// TIA Portal project "XSFW_TIA31001_A0_V15.1" (V15.1)

(* hardware
DEVICE "S7-1200 station_1"  S7-1200 Station
   slot 0: "Rack_0"  S7-1200 Rack  Rack  V1.0
   slot 1: "PLC_Divider"  CPU 1214C DC/DC/DC  6ES7 214-1AG40-0XB0  V4.2
   slot 2: "DI 16/DQ 16x24VDC_1"  6ES7 223-1BL32-0XB0  V2.0
   slot 3: "AI 4x13BIT/AQ 2x14BIT_1"  6ES7 234-4HE32-0XB0  V2.0
   slot 101: "CM 1243-5"  CM 1243-5  6GK7 243-5DX30-0XE0  V1.3
DEVICE "CSM"  SCALANCE X-Station
   slot 0: "Bastidor SCALANCE X"  Rail
   slot 0: "Switch"  6GK7 277-1AA00-0AA0
DEVICE "HMI_1"  KTP700 Basic PN
   slot 0: "HMI_1"  KTP700 Basic PN  6AV2 123-2GB03-0AX0  15.0.0.0
   slot 1: "HMI_RT_1"  KTP700 Basic PN  6AV2 123-2GB03-0AX0  15.0.0.0
   slot 5: "HMI_1.IE_CP_1"  PROFINET Interface  15.0.0.0
      slot 1: "Interfaz PROFINET_1"  PROFINET Interface
         slot 1: "Port_1"  Port
DEVICE "Dispositivo GSD_1"  GSD.Device.PN
   slot 0: "Rack"  Rack  V1.0
   slot 0: "V90-X"  SINAMICS V90 PN V1.0  6SL3 210-5Fxxx-xxFx  V1.00
      slot 0: "SINAMICS V90 PN V1.0"  SINAMICS V90 PN V1.0
      slot 1: "PN-IO"  PN-IO
         slot 1: "Puerto 1"  Port 1
         slot 2: "Puerto 2"  Port 2
      slot 1: "Drive"  Drive
         slot 0: "Punto de acceso a módulo"  Module Access Point
         slot 1: "sin PROFIsafe"  without PROFIsafe
   slot 2: "Telegrama estándar 3, PZD-5/9"  Standard telegram 3, PZD-5/9
DEVICE "Dispositivo GSD_2"  GSD.Device.PN
   slot 0: "Rack"  Rack  V1.0
   slot 0: "V90-Y"  SINAMICS V90 PN V1.0  6SL3 210-5Fxxx-xxFx  V1.00
      slot 0: "SINAMICS V90 PN V1.0"  SINAMICS V90 PN V1.0
      slot 1: "PN-IO"  PN-IO
         slot 1: "Puerto 1"  Port 1
         slot 2: "Puerto 2"  Port 2
      slot 1: "Drive"  Drive
         slot 0: "Punto de acceso a módulo"  Module Access Point
         slot 1: "sin PROFIsafe"  without PROFIsafe
   slot 2: "Telegrama estándar 3, PZD-5/9"  Standard telegram 3, PZD-5/9
*)

// ===== PLC "PLC_Divider"  CPU 1214C DC/DC/DC =====

VAR_GLOBAL   // PLC tag table "Tabla de variables estándar"
   "iCntBot" AT %I0.3 : Bool;
   "iSnsBotBaj" AT %I0.4 : Bool;
   "iSnsBotAlt" AT %I0.5 : Bool;
   "iCH_A" AT %I0.0 : Bool;
   "iCH_B" AT %I0.1 : Bool;
   "iCH_Z" AT %I0.2 : Bool;
   "iSns_Ch1Full" AT %I2.5 : Bool;
   "iSns_Ch2Full" AT %I2.6 : Bool;
   "iSns_Ch3Full" AT %I2.7 : Bool;
   "iSign_HabInv" AT %I3.0 : Bool;
   "iPul_Marcha" AT %I3.1 : Bool;
   "iPul_Parada" AT %I3.2 : Bool;
   "iPul_Rst" AT %I3.3 : Bool;
   "iProt_Abiertas" AT %I3.4 : Bool;
   "iTrip_Inverter" AT %I3.5 : Bool;
   "iRef_Analog" AT %IW54 : Int;
   "qRev_Alarma" AT %Q0.0 : Bool;
   "qSem_Verde" AT %Q0.1 : Bool;
   "qSem_rojo" AT %Q0.2 : Bool;
   "qTest_Marcha" AT %Q0.3 : Bool;
   "qRes_Alarma" AT %Q0.4 : Bool;
   "qRes_Inversor" AT %Q0.5 : Bool;
   "qFwd_Inversor" AT %Q0.6 : Bool;
   "qTrig_2" AT %Q0.7 : Bool;
   "qSign_Marcha" AT %Q1.0 : Bool;
   "qSign_Falla" AT %Q1.1 : Bool;
   "qTrig_1" AT %Q2.0 : Bool;
   "qTrig_22" AT %Q2.1 : Bool;
   "qRef_Analog" AT %IW82 : Int;
   "System_Byte" AT %MB1 : Byte;
   "FirstScan" AT %M1.0 : Bool;
   "DiagStatusUpdate" AT %M1.1 : Bool;
   "AlwaysTRUE" AT %M1.2 : Bool;
   "AlwaysFALSE" AT %M1.3 : Bool;
   "Clock_Byte" AT %MB0 : Byte;
   "Clock_10Hz" AT %M0.0 : Bool;
   "Clock_5Hz" AT %M0.1 : Bool;
   "Clock_2.5Hz" AT %M0.2 : Bool;
   "Clock_2Hz" AT %M0.3 : Bool;
   "Clock_1.25Hz" AT %M0.4 : Bool;
   "Clock_1Hz" AT %M0.5 : Bool;
   "Clock_0.625Hz" AT %M0.6 : Bool;
   "Clock_0.5Hz" AT %M0.7 : Bool;
   "Trip_Inverter" AT %M100.2 : Bool;
   "Marca_Homing" AT %M102.1 : Bool;
   "Eje_X_Drive_IN" AT %I68.0 : "PD_TEL1_IN";
   "Eje_X_Drive_OUT" AT %Q84.0 : "PD_TEL1_OUT";
   "Eje_X_Encoder_IN" AT %I68.0 : "PD_TEL81_IN";
   "Eje_X_Encoder_OUT" AT %Q84.0 : "PD_TEL81_OUT";
   "Eje_Y_Drive_IN" AT %I104.0 : "PD_TEL3_IN";
   "Eje_Y_Drive_OUT" AT %Q74.0 : "PD_TEL3_OUT";
   "Eje_1_Drive_IN" AT %I68.0 : "PD_TEL3_IN";
   "Eje_1_Drive_OUT" AT %Q64.0 : "PD_TEL3_OUT";
END_VAR

VAR_GLOBAL   // PLC tag table "Alarmas"
   "Alarmas_1" AT %MW100 : Word;
   "ProteccionAbierta" AT %M100.0 : Bool;   // Señal I3.4 en 1
   "BotellaCaida" AT %M100.1 : Bool;
END_VAR

VAR_GLOBAL   // PLC tag table "Inicializaciòn"
   "Marcas para la inicializaciòn" AT %MW102 : Word;
   "Start" AT %M102.0 : Bool;
END_VAR

DATA_BLOCK "01_LINEA_Entradas-DB"   // DB1
{ S7_Optimized_Access := 'TRUE' }
VERSION : 0.1
   VAR
      Contador : Bool;   // Pulsador de marcha
      Sensor_Bajo : Bool;   // Pulsador de parada
      Sensor_Alto : Bool;   // Pulsador de marcha columna 4
      CH_A : Bool;   // Pulsador de parada de emergancia columna 4
      CH_B : Bool;   // Pulsador de marcha columna 6
      CH_Z : Bool;   // Pulsador de parada de emergancia columna 6
      Canal1_Full : Bool;   // Pulsador de marcha columna 9
      Canal2_Full : Bool;   // Pulsador de parada de emergancia columna 9
      Canal3_Full : Bool;   // Pulsador de marcha columna 11
      Hab_Inverter : Bool;   // Pulsador de parada de emergancia columna 11
      Marcha : Bool;   // Pulsador de marcha columna 12
      Parada : Bool;   // Pulsador de parada de emergancia columna 12
      Reset : Bool;   // Pulsador de parada de emergancia del tablero general
      Protecciones_Abiertas : Bool;   // Pulsador de parada de emergencia del tablero de la fosa
      Trip_Inverter : Bool;   // Señal de falla del variador
   END_VAR
BEGIN
END_DATA_BLOCK

DATA_BLOCK "02_LINEA_Salidas-DB"   // DB2
{ S7_Optimized_Access := 'TRUE' }
VERSION : 0.1
   VAR
      Alarma_Sonora : Bool;   // Marcha para el variador
      Semaforo_Verde : Bool;   // Sentido adelante variador
      Semaforo_Rojo : Bool;   // Sentido atras variador
      Testigo_Marcha : Bool;   // Indicador sonoro
      Reset_Alarma : Bool;   // Indicador de linea en marcha
      Reset_Inverter : Bool;   // Indicador de linea parada
      Avance_Inverter : Bool;   // Buzzer de la baliza del tablero principal
      Trigger_2 : Bool;   // Lampara verde de la baliza del tablero principal
      EnMarcha : Bool;   // Lampara roja de la baliza del tablero principal
      EnFalla : Bool;   // Lampara amarilla de la baliza del tablero principal
      Trigger_11 : Bool;
      Trigger_22 : Bool;
      Ref_20mA : Int;
   END_VAR
BEGIN
END_DATA_BLOCK

DATA_BLOCK "MotorInverter"   // DB5
{ S7_Optimized_Access := 'TRUE' }
VERSION : 0.1
// stored: InstanceOfName Motor Simple
"Motor Simple"
BEGIN
END_DATA_BLOCK

DATA_BLOCK "Cuentas_Matematicas1_DB"   // DB15
{ S7_Optimized_Access := 'TRUE' }
VERSION : 0.1
   VAR
      MovXNeg : Real := 0.0;
      Mov2X : Real := 0.0;
      Mov2XNeg : Real := 0.0;
      MovYNeg : Real := 0.0;
   END_VAR
BEGIN
END_DATA_BLOCK

DATA_BLOCK "FB_GENERAL_DB"   // DB17
{ S7_Optimized_Access := 'FALSE' }
VERSION : 0.1
// stored: InstanceOfName FB_GENERAL
"FB_GENERAL"
BEGIN
END_DATA_BLOCK

DATA_BLOCK "DB_GENERAL"   // DB100
{ S7_Optimized_Access := 'FALSE' }
VERSION : 0.1
// stored: InstanceOfName FB_GENERAL
"FB_GENERAL"
BEGIN
END_DATA_BLOCK

// folder: COMANDOS

DATA_BLOCK "DB_SUB_0_COM_GENERAL"   // DB600
{ S7_Optimized_Access := 'FALSE' }
VERSION : 0.1
   VAR
      ManipEsperaCarro : Bool;
      RecepCarroConfir : Bool;
      SalidaEsperaCarro1 : Bool;
      SalidaEsperaCarro2 : Bool;
      TengoCarroEnPortacarro : Bool;
      ReconocimientoAlarmas : Bool;
   END_VAR
BEGIN
END_DATA_BLOCK

// folder: INCIDENTES

DATA_BLOCK "DB_INC_GENERAL"   // DB500
{ S7_Optimized_Access := 'FALSE' }
VERSION : 0.1
// stored: InstanceOfName FB_INC_GENERAL
"FB_INC_GENERAL"
BEGIN
END_DATA_BLOCK

// folder: PUESTA EN MARCHA

DATA_BLOCK "DB_PUESTA_MARCHA"   // DB10
{ S7_Optimized_Access := 'TRUE' }
VERSION : 0.1
   VAR
      MovYmm : Real;
      MovXmm : Real;
      TChFull : Time := T#1S;
   END_VAR
BEGIN
END_DATA_BLOCK

// folder: System blocks/Program resources

DATA_BLOCK "IEC_Counter_0_DB"   // DB6
{ S7_Optimized_Access := 'TRUE' }
AUTHOR : Simatic
FAMILY : IEC
NAME : CNTR
VERSION : 1.0
// stored: InstanceOfName IEC_COUNTER
"IEC_COUNTER"
BEGIN
END_DATA_BLOCK

DATA_BLOCK "IEC_Timer_0_DB"   // DB7
{ S7_Optimized_Access := 'TRUE' }
AUTHOR : Simatic
FAMILY : IEC
NAME : IEC_TMR
VERSION : 1.0
// stored: InstanceOfName IEC_TIMER
"IEC_TIMER"
BEGIN
END_DATA_BLOCK

DATA_BLOCK "IEC_Counter_1_DB"   // DB8
{ S7_Optimized_Access := 'TRUE' }
AUTHOR : Simatic
FAMILY : IEC
NAME : CNTR
VERSION : 1.0
// stored: InstanceOfName IEC_COUNTER
"IEC_COUNTER"
BEGIN
END_DATA_BLOCK

DATA_BLOCK "IEC_Counter_2_DB"   // DB9
{ S7_Optimized_Access := 'TRUE' }
AUTHOR : Simatic
FAMILY : IEC
NAME : CNTR
VERSION : 1.0
// stored: InstanceOfName IEC_COUNTER
"IEC_COUNTER"
BEGIN
END_DATA_BLOCK

DATA_BLOCK "IEC_Timer_ChFull"   // DB11
{ S7_Optimized_Access := 'TRUE' }
AUTHOR : Simatic
FAMILY : IEC
NAME : IEC_TMR
VERSION : 1.0
// stored: InstanceOfName IEC_TIMER
"IEC_TIMER"
BEGIN
END_DATA_BLOCK

// folder: VISUALIZACION

DATA_BLOCK "DB_VIS_GENERAL"   // DB800
{ S7_Optimized_Access := 'FALSE' }
VERSION : 0.1
   VAR
      CantBot : Int;
      AlarmaProtecciòn : Bool;
      AlarmaBotellaCaida : Bool;
      Homing : Bool;
   END_VAR
BEGIN
END_DATA_BLOCK

// folder: (top level)

DATA_BLOCK "Eje_Y"   // DB4, Motion_DB
{ S7_Optimized_Access := 'TRUE' }
AUTHOR : SIMATIC
FAMILY : BasicMC
NAME : TO_PosAx
VERSION : 6.0
// stored: InstanceOfName TO_PositioningAxis
"TO_PositioningAxis"
BEGIN
   // Axis.Encoder.TelegramAddressOutCU = %Q74.0
   // Axis.Encoder.TelegramAddressInCU = %I104.0
   // Axis.Encoder.DoNameCU = V90-Y.Drive_Encóder1
   // Axis.Drive.TelegramAddressOutCU = %Q74.0
   // Axis.Drive.TelegramAddressInCU = %I104.0
   // Axis.Drive.TelegramType = 2
   // Axis.Drive.DoNameCU = V90-Y.Drive
   // Axis.LengthUnitNormalized.Time = 1
   // Axis.LengthUnitNormalized.Distance = -2
   // Axis.Encoder.SelectedHscIndexCU = -1
   // Axis.Encoder.DbTypeCU = Classic
   // Axis.Drive.DbTypeCU = Classic
END_DATA_BLOCK

DATA_BLOCK "Eje_X"   // DB12, Motion_DB
{ S7_Optimized_Access := 'TRUE' }
AUTHOR : SIMATIC
FAMILY : BasicMC
NAME : TO_PosAx
VERSION : 6.0
// stored: InstanceOfName TO_PositioningAxis
"TO_PositioningAxis"
BEGIN
   // Axis.Encoder.TelegramAddressOutCU = %Q64.0
   // Axis.Encoder.TelegramAddressInCU = %I68.0
   // Axis.Encoder.DoNameCU = V90-X.Drive_Encóder1
   // Axis.Drive.TelegramAddressOutCU = %Q64.0
   // Axis.Drive.TelegramAddressInCU = %I68.0
   // Axis.Drive.TelegramType = 2
   // Axis.Drive.DoNameCU = V90-X.Drive
   // Axis.LengthUnitNormalized.Distance = 1013
   // Axis.Encoder.SelectedHscIndexCU = -1
   // Axis.Encoder.DbTypeCU = Classic
   // Axis.Drive.DbTypeCU = Classic
END_DATA_BLOCK

FUNCTION_BLOCK "Cuentas_Matematicas1"   // FB1, LAD
{ S7_Optimized_Access := 'TRUE' }
VERSION : 0.1
BEGIN

REGION Network 1: Movimiento negativo en X
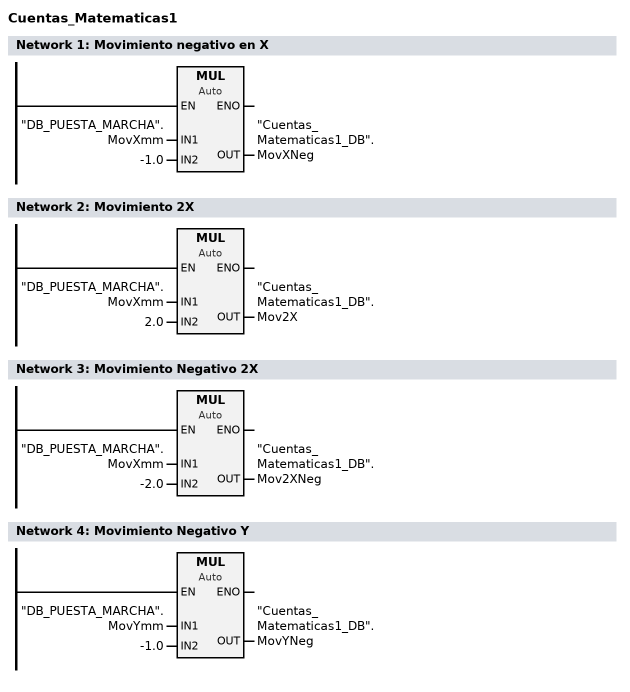
   RUNG wire#powerrail
      Mul(in1 := "DB_PUESTA_MARCHA".MovXmm, in2 := -1.0, out => "Cuentas_Matematicas1_DB".MovXNeg)
   END_RUNG
   // the same network as SCL:
   "Cuentas_Matematicas1_DB".MovXNeg := "DB_PUESTA_MARCHA".MovXmm * (-1.0);
END_REGION

REGION Network 2: Movimiento 2X
   RUNG wire#powerrail
      Mul(in1 := "DB_PUESTA_MARCHA".MovXmm, in2 := 2.0, out => "Cuentas_Matematicas1_DB".Mov2X)
   END_RUNG
   // the same network as SCL:
   "Cuentas_Matematicas1_DB".Mov2X := "DB_PUESTA_MARCHA".MovXmm * 2.0;
END_REGION

REGION Network 3: Movimiento Negativo 2X
   RUNG wire#powerrail
      Mul(in1 := "DB_PUESTA_MARCHA".MovXmm, in2 := -2.0, out => "Cuentas_Matematicas1_DB".Mov2XNeg)
   END_RUNG
   // the same network as SCL:
   "Cuentas_Matematicas1_DB".Mov2XNeg := "DB_PUESTA_MARCHA".MovXmm * (-2.0);
END_REGION

REGION Network 4: Movimiento Negativo Y
   RUNG wire#powerrail
      Mul(in1 := "DB_PUESTA_MARCHA".MovYmm, in2 := -1.0, out => "Cuentas_Matematicas1_DB".MovYNeg)
   END_RUNG
   // the same network as SCL:
   "Cuentas_Matematicas1_DB".MovYNeg := "DB_PUESTA_MARCHA".MovYmm * (-1.0);
END_REGION
END_FUNCTION_BLOCK

FUNCTION_BLOCK "FB_GENERAL"   // FB100, LAD
{ S7_Optimized_Access := 'FALSE' }
VERSION : 0.1
   VAR_OUTPUT
      DoneX : Bool;
      DoneY : Bool;
      Done2X : Bool;
      DoneHomeX : Bool;
      DoneHomeY : Bool;
   END_VAR
   VAR
      Estados : Array[0..32] of Bool;
      Concatenadoras : Array[0..32] of Bool;
      Prioritarias : Array[0..32] of Bool;
      Error_Concatenadoras : Bool;
      Error_Prioritarias : Bool;
      Cuenta_1 : Bool;
      Cuenta_2 : Bool;
      Cuenta_3 : Bool;
      "Cont_Botellas/2" : Int;
   END_VAR
BEGIN

REGION Network 1: Inicializaciòn
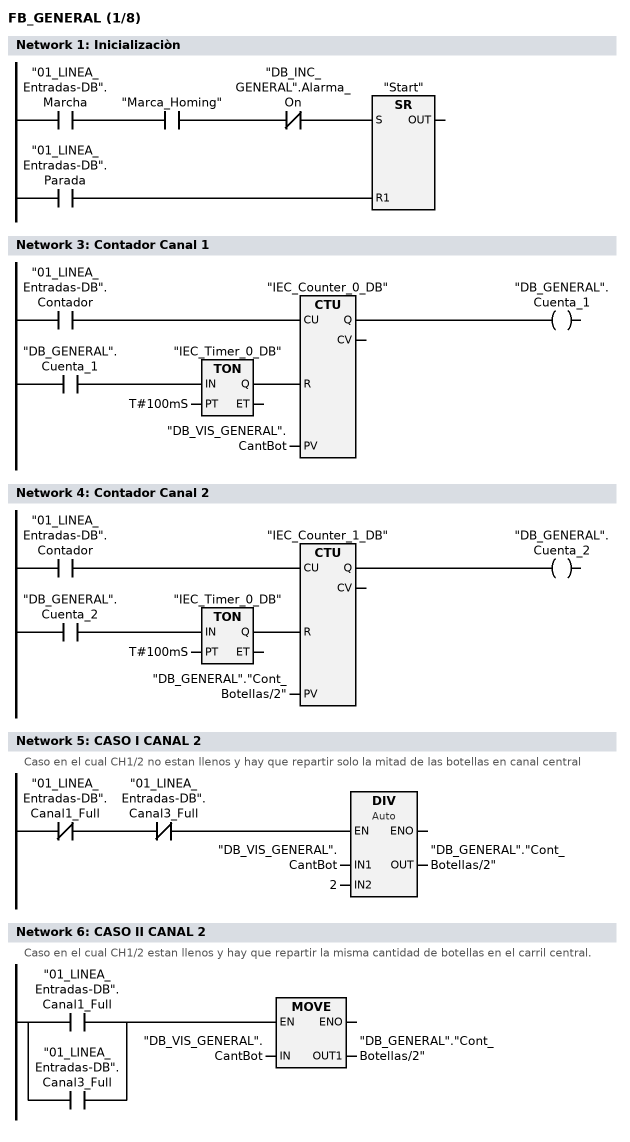
   RUNG wire#powerrail
      Contact( "01_LINEA_Entradas-DB".Marcha )
      Contact( "Marca_Homing" )
      I_Contact( "DB_INC_GENERAL".Alarma_On )
      S_SR(operand := "Start", r1 := wire#w1)
   END_RUNG
   RUNG wire#powerrail
      Contact( "01_LINEA_Entradas-DB".Parada )
   END_RUNG wire#w1
   // the same network as SCL:
   IF "01_LINEA_Entradas-DB".Marcha AND "Marca_Homing" AND NOT "DB_INC_GENERAL".Alarma_On THEN
       "Start" := TRUE;   // SR flip-flop
   END_IF;
   IF "01_LINEA_Entradas-DB".Parada THEN "Start" := FALSE; END_IF;
END_REGION

REGION Network 2: -----------------OTROS---------------
END_REGION

REGION Network 3: Contador Canal 1
   "IEC_Timer_0_DB".TON(IN := "DB_GENERAL".Cuenta_1, PT := T#100mS);
   "IEC_Counter_0_DB".CTU(CU := "01_LINEA_Entradas-DB".Contador,
                          R := "IEC_Timer_0_DB".Q,
                          PV := "DB_VIS_GENERAL".CantBot);
   "DB_GENERAL".Cuenta_1 := "IEC_Counter_0_DB".Q;
END_REGION

REGION Network 4: Contador Canal 2
   "IEC_Timer_0_DB".TON(IN := "DB_GENERAL".Cuenta_2, PT := T#100mS);
   "IEC_Counter_1_DB".CTU(CU := "01_LINEA_Entradas-DB".Contador,
                          R := "IEC_Timer_0_DB".Q,
                          PV := "DB_GENERAL"."Cont_Botellas/2");
   "DB_GENERAL".Cuenta_2 := "IEC_Counter_1_DB".Q;
END_REGION

REGION Network 5: CASO I CANAL 2
   // Caso en el cual CH1/2 no estan llenos y hay que repartir solo la mitad de las botellas en canal central
   RUNG wire#powerrail
      I_Contact( "01_LINEA_Entradas-DB".Canal1_Full )
      I_Contact( "01_LINEA_Entradas-DB".Canal3_Full )
      Div(in1 := "DB_VIS_GENERAL".CantBot, in2 := 2, out => "DB_GENERAL"."Cont_Botellas/2")
   END_RUNG
   // the same network as SCL:
   IF NOT "01_LINEA_Entradas-DB".Canal1_Full AND NOT "01_LINEA_Entradas-DB".Canal3_Full THEN
       "DB_GENERAL"."Cont_Botellas/2" := "DB_VIS_GENERAL".CantBot / 2;
   END_IF;
END_REGION

REGION Network 6: CASO II CANAL 2
   // Caso en el cual CH1/2 estan llenos y hay que repartir la misma cantidad de botellas en el carril central.
   RUNG wire#powerrail
      Contact( "01_LINEA_Entradas-DB".Canal1_Full )
      wire#w1
      Move(in := "DB_VIS_GENERAL".CantBot, out1 => "DB_GENERAL"."Cont_Botellas/2")
   END_RUNG
   RUNG wire#powerrail
      Contact( "01_LINEA_Entradas-DB".Canal3_Full )
   END_RUNG wire#w1
   // the same network as SCL:
   IF "01_LINEA_Entradas-DB".Canal1_Full OR "01_LINEA_Entradas-DB".Canal3_Full THEN
       "DB_GENERAL"."Cont_Botellas/2" := "DB_VIS_GENERAL".CantBot;
   END_IF;
END_REGION

REGION Network 7: Contador Canal 3
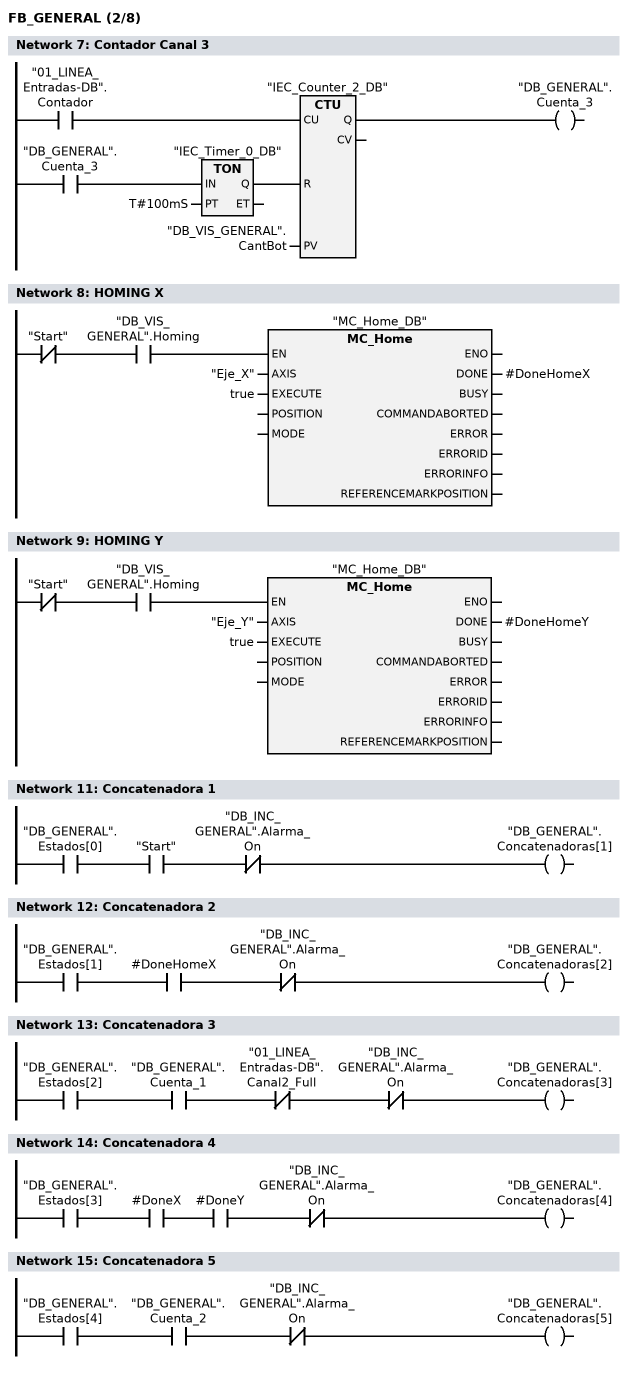
   "IEC_Timer_0_DB".TON(IN := "DB_GENERAL".Cuenta_3, PT := T#100mS);
   "IEC_Counter_2_DB".CTU(CU := "01_LINEA_Entradas-DB".Contador,
                          R := "IEC_Timer_0_DB".Q,
                          PV := "DB_VIS_GENERAL".CantBot);
   "DB_GENERAL".Cuenta_3 := "IEC_Counter_2_DB".Q;
END_REGION

REGION Network 8: HOMING X
   IF NOT "Start" AND "DB_VIS_GENERAL".Homing THEN
       "MC_Home_DB"(Axis := "Eje_X", Execute := true, Done => #DoneHomeX);   // MC_Home
   END_IF;
END_REGION

REGION Network 9: HOMING Y
   IF NOT "Start" AND "DB_VIS_GENERAL".Homing THEN
       "MC_Home_DB"(Axis := "Eje_Y", Execute := true, Done => #DoneHomeY);   // MC_Home
   END_IF;
END_REGION

REGION Network 10: --------------------Maquina de estados - 3 carriles-----------------
END_REGION

REGION Network 11: Concatenadora 1
   RUNG wire#powerrail
      Contact( "DB_GENERAL".Estados[0] )
      Contact( "Start" )
      I_Contact( "DB_INC_GENERAL".Alarma_On )
      Coil( "DB_GENERAL".Concatenadoras[1] )
   END_RUNG
   // the same network as SCL:
   "DB_GENERAL".Concatenadoras[1] := "DB_GENERAL".Estados[0] AND "Start" AND NOT "DB_INC_GENERAL".Alarma_On;
END_REGION

REGION Network 12: Concatenadora 2
   RUNG wire#powerrail
      Contact( "DB_GENERAL".Estados[1] )
      Contact( #DoneHomeX )
      I_Contact( "DB_INC_GENERAL".Alarma_On )
      Coil( "DB_GENERAL".Concatenadoras[2] )
   END_RUNG
   // the same network as SCL:
   "DB_GENERAL".Concatenadoras[2] := "DB_GENERAL".Estados[1] AND #DoneHomeX AND NOT "DB_INC_GENERAL".Alarma_On;
END_REGION

REGION Network 13: Concatenadora 3
   RUNG wire#powerrail
      Contact( "DB_GENERAL".Estados[2] )
      Contact( "DB_GENERAL".Cuenta_1 )
      I_Contact( "01_LINEA_Entradas-DB".Canal2_Full )
      I_Contact( "DB_INC_GENERAL".Alarma_On )
      Coil( "DB_GENERAL".Concatenadoras[3] )
   END_RUNG
   // the same network as SCL:
   "DB_GENERAL".Concatenadoras[3] := "DB_GENERAL".Estados[2] AND "DB_GENERAL".Cuenta_1 AND NOT "01_LINEA_Entradas-DB".Canal2_Full AND NOT "DB_INC_GENERAL".Alarma_On;
END_REGION

REGION Network 14: Concatenadora 4
   RUNG wire#powerrail
      Contact( "DB_GENERAL".Estados[3] )
      Contact( #DoneX )
      Contact( #DoneY )
      I_Contact( "DB_INC_GENERAL".Alarma_On )
      Coil( "DB_GENERAL".Concatenadoras[4] )
   END_RUNG
   // the same network as SCL:
   "DB_GENERAL".Concatenadoras[4] := "DB_GENERAL".Estados[3] AND #DoneX AND #DoneY AND NOT "DB_INC_GENERAL".Alarma_On;
END_REGION

REGION Network 15: Concatenadora 5
   RUNG wire#powerrail
      Contact( "DB_GENERAL".Estados[4] )
      Contact( "DB_GENERAL".Cuenta_2 )
      I_Contact( "DB_INC_GENERAL".Alarma_On )
      Coil( "DB_GENERAL".Concatenadoras[5] )
   END_RUNG
   // the same network as SCL:
   "DB_GENERAL".Concatenadoras[5] := "DB_GENERAL".Estados[4] AND "DB_GENERAL".Cuenta_2 AND NOT "DB_INC_GENERAL".Alarma_On;
END_REGION

REGION Network 16: Concatenadora 6
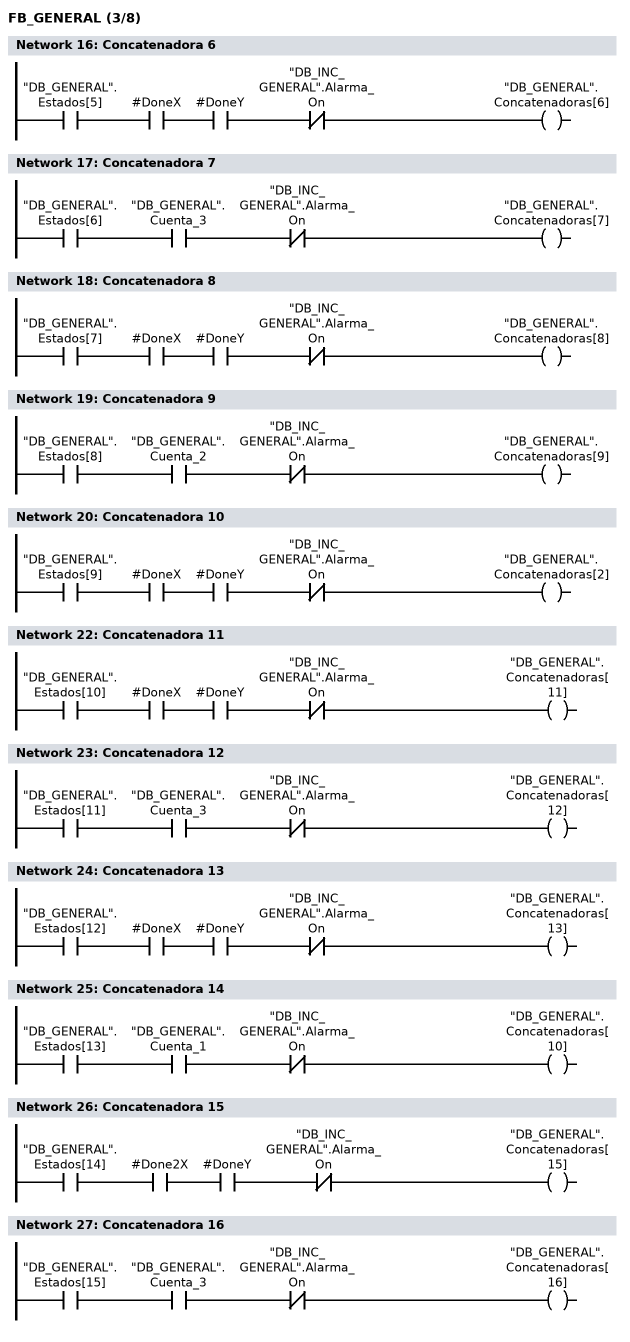
   RUNG wire#powerrail
      Contact( "DB_GENERAL".Estados[5] )
      Contact( #DoneX )
      Contact( #DoneY )
      I_Contact( "DB_INC_GENERAL".Alarma_On )
      Coil( "DB_GENERAL".Concatenadoras[6] )
   END_RUNG
   // the same network as SCL:
   "DB_GENERAL".Concatenadoras[6] := "DB_GENERAL".Estados[5] AND #DoneX AND #DoneY AND NOT "DB_INC_GENERAL".Alarma_On;
END_REGION

REGION Network 17: Concatenadora 7
   RUNG wire#powerrail
      Contact( "DB_GENERAL".Estados[6] )
      Contact( "DB_GENERAL".Cuenta_3 )
      I_Contact( "DB_INC_GENERAL".Alarma_On )
      Coil( "DB_GENERAL".Concatenadoras[7] )
   END_RUNG
   // the same network as SCL:
   "DB_GENERAL".Concatenadoras[7] := "DB_GENERAL".Estados[6] AND "DB_GENERAL".Cuenta_3 AND NOT "DB_INC_GENERAL".Alarma_On;
END_REGION

REGION Network 18: Concatenadora 8
   RUNG wire#powerrail
      Contact( "DB_GENERAL".Estados[7] )
      Contact( #DoneX )
      Contact( #DoneY )
      I_Contact( "DB_INC_GENERAL".Alarma_On )
      Coil( "DB_GENERAL".Concatenadoras[8] )
   END_RUNG
   // the same network as SCL:
   "DB_GENERAL".Concatenadoras[8] := "DB_GENERAL".Estados[7] AND #DoneX AND #DoneY AND NOT "DB_INC_GENERAL".Alarma_On;
END_REGION

REGION Network 19: Concatenadora 9
   RUNG wire#powerrail
      Contact( "DB_GENERAL".Estados[8] )
      Contact( "DB_GENERAL".Cuenta_2 )
      I_Contact( "DB_INC_GENERAL".Alarma_On )
      Coil( "DB_GENERAL".Concatenadoras[9] )
   END_RUNG
   // the same network as SCL:
   "DB_GENERAL".Concatenadoras[9] := "DB_GENERAL".Estados[8] AND "DB_GENERAL".Cuenta_2 AND NOT "DB_INC_GENERAL".Alarma_On;
END_REGION

REGION Network 20: Concatenadora 10
   RUNG wire#powerrail
      Contact( "DB_GENERAL".Estados[9] )
      Contact( #DoneX )
      Contact( #DoneY )
      I_Contact( "DB_INC_GENERAL".Alarma_On )
      Coil( "DB_GENERAL".Concatenadoras[2] )
   END_RUNG
   // the same network as SCL:
   "DB_GENERAL".Concatenadoras[2] := "DB_GENERAL".Estados[9] AND #DoneX AND #DoneY AND NOT "DB_INC_GENERAL".Alarma_On;
END_REGION

REGION Network 21: ---------------Maquina de estado - 2 carriles -------------
END_REGION

REGION Network 22: Concatenadora 11
   RUNG wire#powerrail
      Contact( "DB_GENERAL".Estados[10] )
      Contact( #DoneX )
      Contact( #DoneY )
      I_Contact( "DB_INC_GENERAL".Alarma_On )
      Coil( "DB_GENERAL".Concatenadoras[11] )
   END_RUNG
   // the same network as SCL:
   "DB_GENERAL".Concatenadoras[11] := "DB_GENERAL".Estados[10] AND #DoneX AND #DoneY AND NOT "DB_INC_GENERAL".Alarma_On;
END_REGION

REGION Network 23: Concatenadora 12
   RUNG wire#powerrail
      Contact( "DB_GENERAL".Estados[11] )
      Contact( "DB_GENERAL".Cuenta_3 )
      I_Contact( "DB_INC_GENERAL".Alarma_On )
      Coil( "DB_GENERAL".Concatenadoras[12] )
   END_RUNG
   // the same network as SCL:
   "DB_GENERAL".Concatenadoras[12] := "DB_GENERAL".Estados[11] AND "DB_GENERAL".Cuenta_3 AND NOT "DB_INC_GENERAL".Alarma_On;
END_REGION

REGION Network 24: Concatenadora 13
   RUNG wire#powerrail
      Contact( "DB_GENERAL".Estados[12] )
      Contact( #DoneX )
      Contact( #DoneY )
      I_Contact( "DB_INC_GENERAL".Alarma_On )
      Coil( "DB_GENERAL".Concatenadoras[13] )
   END_RUNG
   // the same network as SCL:
   "DB_GENERAL".Concatenadoras[13] := "DB_GENERAL".Estados[12] AND #DoneX AND #DoneY AND NOT "DB_INC_GENERAL".Alarma_On;
END_REGION

REGION Network 25: Concatenadora 14
   RUNG wire#powerrail
      Contact( "DB_GENERAL".Estados[13] )
      Contact( "DB_GENERAL".Cuenta_1 )
      I_Contact( "DB_INC_GENERAL".Alarma_On )
      Coil( "DB_GENERAL".Concatenadoras[10] )
   END_RUNG
   // the same network as SCL:
   "DB_GENERAL".Concatenadoras[10] := "DB_GENERAL".Estados[13] AND "DB_GENERAL".Cuenta_1 AND NOT "DB_INC_GENERAL".Alarma_On;
END_REGION

REGION Network 26: Concatenadora 15
   RUNG wire#powerrail
      Contact( "DB_GENERAL".Estados[14] )
      Contact( #Done2X )
      Contact( #DoneY )
      I_Contact( "DB_INC_GENERAL".Alarma_On )
      Coil( "DB_GENERAL".Concatenadoras[15] )
   END_RUNG
   // the same network as SCL:
   "DB_GENERAL".Concatenadoras[15] := "DB_GENERAL".Estados[14] AND #Done2X AND #DoneY AND NOT "DB_INC_GENERAL".Alarma_On;
END_REGION

REGION Network 27: Concatenadora 16
   RUNG wire#powerrail
      Contact( "DB_GENERAL".Estados[15] )
      Contact( "DB_GENERAL".Cuenta_3 )
      I_Contact( "DB_INC_GENERAL".Alarma_On )
      Coil( "DB_GENERAL".Concatenadoras[16] )
   END_RUNG
   // the same network as SCL:
   "DB_GENERAL".Concatenadoras[16] := "DB_GENERAL".Estados[15] AND "DB_GENERAL".Cuenta_3 AND NOT "DB_INC_GENERAL".Alarma_On;
END_REGION

REGION Network 28: Concatenadora 17
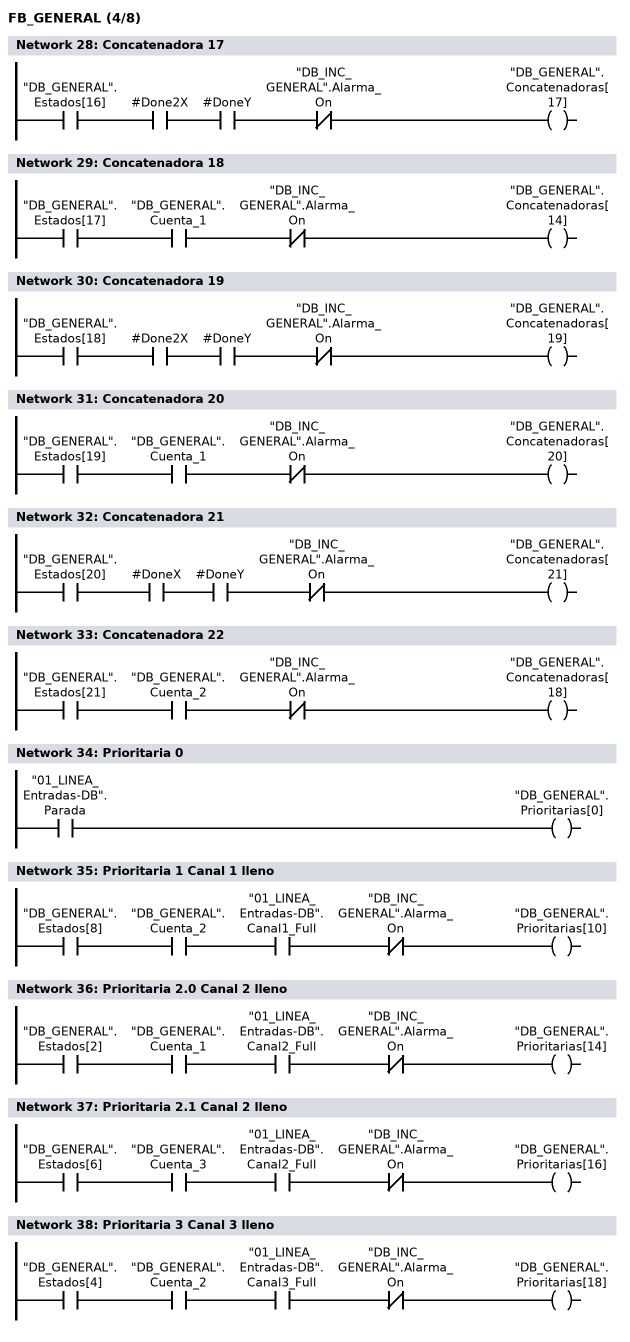
   RUNG wire#powerrail
      Contact( "DB_GENERAL".Estados[16] )
      Contact( #Done2X )
      Contact( #DoneY )
      I_Contact( "DB_INC_GENERAL".Alarma_On )
      Coil( "DB_GENERAL".Concatenadoras[17] )
   END_RUNG
   // the same network as SCL:
   "DB_GENERAL".Concatenadoras[17] := "DB_GENERAL".Estados[16] AND #Done2X AND #DoneY AND NOT "DB_INC_GENERAL".Alarma_On;
END_REGION

REGION Network 29: Concatenadora 18
   RUNG wire#powerrail
      Contact( "DB_GENERAL".Estados[17] )
      Contact( "DB_GENERAL".Cuenta_1 )
      I_Contact( "DB_INC_GENERAL".Alarma_On )
      Coil( "DB_GENERAL".Concatenadoras[14] )
   END_RUNG
   // the same network as SCL:
   "DB_GENERAL".Concatenadoras[14] := "DB_GENERAL".Estados[17] AND "DB_GENERAL".Cuenta_1 AND NOT "DB_INC_GENERAL".Alarma_On;
END_REGION

REGION Network 30: Concatenadora 19
   RUNG wire#powerrail
      Contact( "DB_GENERAL".Estados[18] )
      Contact( #Done2X )
      Contact( #DoneY )
      I_Contact( "DB_INC_GENERAL".Alarma_On )
      Coil( "DB_GENERAL".Concatenadoras[19] )
   END_RUNG
   // the same network as SCL:
   "DB_GENERAL".Concatenadoras[19] := "DB_GENERAL".Estados[18] AND #Done2X AND #DoneY AND NOT "DB_INC_GENERAL".Alarma_On;
END_REGION

REGION Network 31: Concatenadora 20
   RUNG wire#powerrail
      Contact( "DB_GENERAL".Estados[19] )
      Contact( "DB_GENERAL".Cuenta_1 )
      I_Contact( "DB_INC_GENERAL".Alarma_On )
      Coil( "DB_GENERAL".Concatenadoras[20] )
   END_RUNG
   // the same network as SCL:
   "DB_GENERAL".Concatenadoras[20] := "DB_GENERAL".Estados[19] AND "DB_GENERAL".Cuenta_1 AND NOT "DB_INC_GENERAL".Alarma_On;
END_REGION

REGION Network 32: Concatenadora 21
   RUNG wire#powerrail
      Contact( "DB_GENERAL".Estados[20] )
      Contact( #DoneX )
      Contact( #DoneY )
      I_Contact( "DB_INC_GENERAL".Alarma_On )
      Coil( "DB_GENERAL".Concatenadoras[21] )
   END_RUNG
   // the same network as SCL:
   "DB_GENERAL".Concatenadoras[21] := "DB_GENERAL".Estados[20] AND #DoneX AND #DoneY AND NOT "DB_INC_GENERAL".Alarma_On;
END_REGION

REGION Network 33: Concatenadora 22
   RUNG wire#powerrail
      Contact( "DB_GENERAL".Estados[21] )
      Contact( "DB_GENERAL".Cuenta_2 )
      I_Contact( "DB_INC_GENERAL".Alarma_On )
      Coil( "DB_GENERAL".Concatenadoras[18] )
   END_RUNG
   // the same network as SCL:
   "DB_GENERAL".Concatenadoras[18] := "DB_GENERAL".Estados[21] AND "DB_GENERAL".Cuenta_2 AND NOT "DB_INC_GENERAL".Alarma_On;
END_REGION

REGION Network 34: Prioritaria 0
   RUNG wire#powerrail
      Contact( "01_LINEA_Entradas-DB".Parada )
      Coil( "DB_GENERAL".Prioritarias[0] )
   END_RUNG
   // the same network as SCL:
   "DB_GENERAL".Prioritarias[0] := "01_LINEA_Entradas-DB".Parada;
END_REGION

REGION Network 35: Prioritaria 1 Canal 1 lleno
   RUNG wire#powerrail
      Contact( "DB_GENERAL".Estados[8] )
      Contact( "DB_GENERAL".Cuenta_2 )
      Contact( "01_LINEA_Entradas-DB".Canal1_Full )
      I_Contact( "DB_INC_GENERAL".Alarma_On )
      Coil( "DB_GENERAL".Prioritarias[10] )
   END_RUNG
   // the same network as SCL:
   "DB_GENERAL".Prioritarias[10] := "DB_GENERAL".Estados[8] AND "DB_GENERAL".Cuenta_2 AND "01_LINEA_Entradas-DB".Canal1_Full AND NOT "DB_INC_GENERAL".Alarma_On;
END_REGION

REGION Network 36: Prioritaria 2.0 Canal 2 lleno
   RUNG wire#powerrail
      Contact( "DB_GENERAL".Estados[2] )
      Contact( "DB_GENERAL".Cuenta_1 )
      Contact( "01_LINEA_Entradas-DB".Canal2_Full )
      I_Contact( "DB_INC_GENERAL".Alarma_On )
      Coil( "DB_GENERAL".Prioritarias[14] )
   END_RUNG
   // the same network as SCL:
   "DB_GENERAL".Prioritarias[14] := "DB_GENERAL".Estados[2] AND "DB_GENERAL".Cuenta_1 AND "01_LINEA_Entradas-DB".Canal2_Full AND NOT "DB_INC_GENERAL".Alarma_On;
END_REGION

REGION Network 37: Prioritaria 2.1 Canal 2 lleno
   RUNG wire#powerrail
      Contact( "DB_GENERAL".Estados[6] )
      Contact( "DB_GENERAL".Cuenta_3 )
      Contact( "01_LINEA_Entradas-DB".Canal2_Full )
      I_Contact( "DB_INC_GENERAL".Alarma_On )
      Coil( "DB_GENERAL".Prioritarias[16] )
   END_RUNG
   // the same network as SCL:
   "DB_GENERAL".Prioritarias[16] := "DB_GENERAL".Estados[6] AND "DB_GENERAL".Cuenta_3 AND "01_LINEA_Entradas-DB".Canal2_Full AND NOT "DB_INC_GENERAL".Alarma_On;
END_REGION

REGION Network 38: Prioritaria 3 Canal 3 lleno
   RUNG wire#powerrail
      Contact( "DB_GENERAL".Estados[4] )
      Contact( "DB_GENERAL".Cuenta_2 )
      Contact( "01_LINEA_Entradas-DB".Canal3_Full )
      I_Contact( "DB_INC_GENERAL".Alarma_On )
      Coil( "DB_GENERAL".Prioritarias[18] )
   END_RUNG
   // the same network as SCL:
   "DB_GENERAL".Prioritarias[18] := "DB_GENERAL".Estados[4] AND "DB_GENERAL".Cuenta_2 AND "01_LINEA_Entradas-DB".Canal3_Full AND NOT "DB_INC_GENERAL".Alarma_On;
END_REGION

REGION Network 39: Prioritaria 4 Canal 1 se vaciò
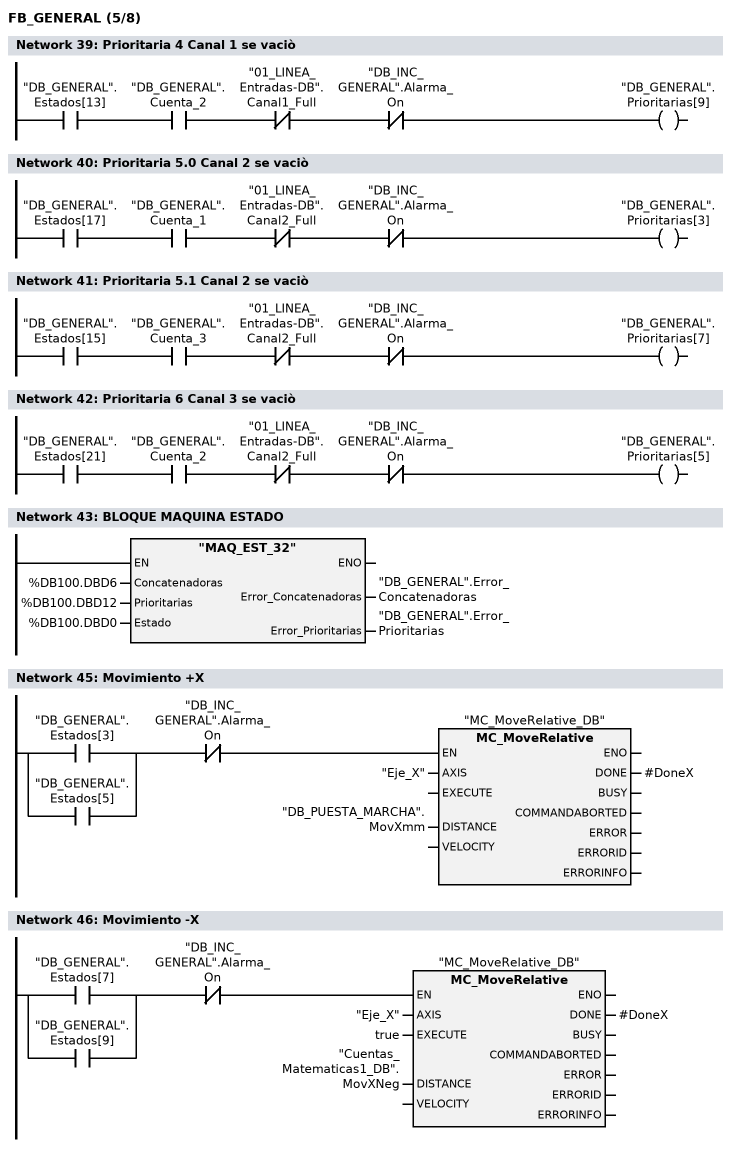
   RUNG wire#powerrail
      Contact( "DB_GENERAL".Estados[13] )
      Contact( "DB_GENERAL".Cuenta_2 )
      I_Contact( "01_LINEA_Entradas-DB".Canal1_Full )
      I_Contact( "DB_INC_GENERAL".Alarma_On )
      Coil( "DB_GENERAL".Prioritarias[9] )
   END_RUNG
   // the same network as SCL:
   "DB_GENERAL".Prioritarias[9] := "DB_GENERAL".Estados[13] AND "DB_GENERAL".Cuenta_2 AND NOT "01_LINEA_Entradas-DB".Canal1_Full AND NOT "DB_INC_GENERAL".Alarma_On;
END_REGION

REGION Network 40: Prioritaria 5.0 Canal 2 se vaciò
   RUNG wire#powerrail
      Contact( "DB_GENERAL".Estados[17] )
      Contact( "DB_GENERAL".Cuenta_1 )
      I_Contact( "01_LINEA_Entradas-DB".Canal2_Full )
      I_Contact( "DB_INC_GENERAL".Alarma_On )
      Coil( "DB_GENERAL".Prioritarias[3] )
   END_RUNG
   // the same network as SCL:
   "DB_GENERAL".Prioritarias[3] := "DB_GENERAL".Estados[17] AND "DB_GENERAL".Cuenta_1 AND NOT "01_LINEA_Entradas-DB".Canal2_Full AND NOT "DB_INC_GENERAL".Alarma_On;
END_REGION

REGION Network 41: Prioritaria 5.1 Canal 2 se vaciò
   RUNG wire#powerrail
      Contact( "DB_GENERAL".Estados[15] )
      Contact( "DB_GENERAL".Cuenta_3 )
      I_Contact( "01_LINEA_Entradas-DB".Canal2_Full )
      I_Contact( "DB_INC_GENERAL".Alarma_On )
      Coil( "DB_GENERAL".Prioritarias[7] )
   END_RUNG
   // the same network as SCL:
   "DB_GENERAL".Prioritarias[7] := "DB_GENERAL".Estados[15] AND "DB_GENERAL".Cuenta_3 AND NOT "01_LINEA_Entradas-DB".Canal2_Full AND NOT "DB_INC_GENERAL".Alarma_On;
END_REGION

REGION Network 42: Prioritaria 6 Canal 3 se vaciò
   RUNG wire#powerrail
      Contact( "DB_GENERAL".Estados[21] )
      Contact( "DB_GENERAL".Cuenta_2 )
      I_Contact( "01_LINEA_Entradas-DB".Canal2_Full )
      I_Contact( "DB_INC_GENERAL".Alarma_On )
      Coil( "DB_GENERAL".Prioritarias[5] )
   END_RUNG
   // the same network as SCL:
   "DB_GENERAL".Prioritarias[5] := "DB_GENERAL".Estados[21] AND "DB_GENERAL".Cuenta_2 AND NOT "01_LINEA_Entradas-DB".Canal2_Full AND NOT "DB_INC_GENERAL".Alarma_On;
END_REGION

REGION Network 43: BLOQUE MAQUINA ESTADO
   RUNG wire#powerrail
      "MAQ_EST_32"(Concatenadoras := %DB100.DBD6, Prioritarias := %DB100.DBD12, Estado := %DB100.DBD0, Error_Concatenadoras => "DB_GENERAL".Error_Concatenadoras, Error_Prioritarias => "DB_GENERAL".Error_Prioritarias)
   END_RUNG
   // the same network as SCL:
   "MAQ_EST_32"(Concatenadoras := %DB100.DBD6,
                Prioritarias := %DB100.DBD12,
                Estado := %DB100.DBD0,
                Error_Concatenadoras => "DB_GENERAL".Error_Concatenadoras,
                Error_Prioritarias => "DB_GENERAL".Error_Prioritarias);
END_REGION

REGION Network 44: --------------ACCIONAMIENTOS----------------
END_REGION

REGION Network 45: Movimiento +X
   IF ("DB_GENERAL".Estados[3] OR "DB_GENERAL".Estados[5]) AND NOT "DB_INC_GENERAL".Alarma_On THEN
       "MC_MoveRelative_DB"(Axis := "Eje_X", Distance := "DB_PUESTA_MARCHA".MovXmm, Done => #DoneX);   // MC_MoveRelative
   END_IF;
END_REGION

REGION Network 46: Movimiento -X
   IF ("DB_GENERAL".Estados[7] OR "DB_GENERAL".Estados[9]) AND NOT "DB_INC_GENERAL".Alarma_On THEN
       "MC_MoveRelative_DB"(Axis := "Eje_X",   // MC_MoveRelative
                            Execute := true,
                            Distance := "Cuentas_Matematicas1_DB".MovXNeg,
                            Done => #DoneX);
   END_IF;
END_REGION

REGION Network 47: Movimiento +Y
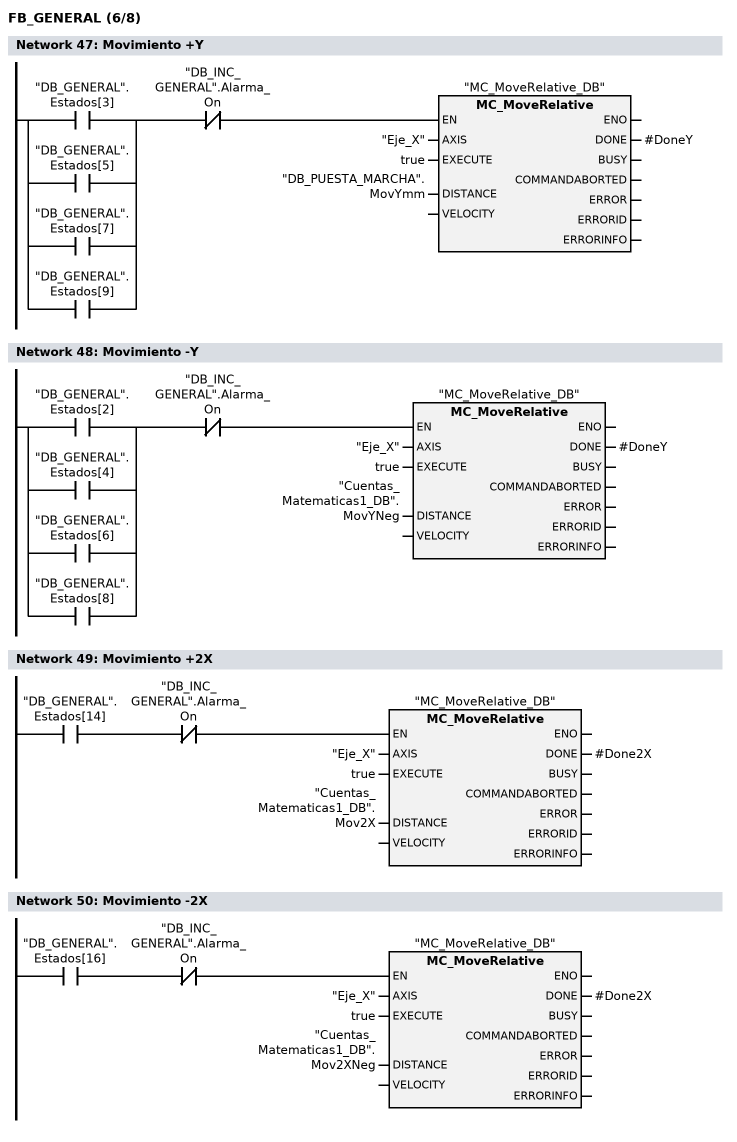
   IF ("DB_GENERAL".Estados[3] OR "DB_GENERAL".Estados[5] OR "DB_GENERAL".Estados[7] OR "DB_GENERAL".Estados[9]) AND NOT "DB_INC_GENERAL".Alarma_On THEN
       "MC_MoveRelative_DB"(Axis := "Eje_X", Execute := true, Distance := "DB_PUESTA_MARCHA".MovYmm, Done => #DoneY);   // MC_MoveRelative
   END_IF;
END_REGION

REGION Network 48: Movimiento -Y
   IF ("DB_GENERAL".Estados[2] OR "DB_GENERAL".Estados[4] OR "DB_GENERAL".Estados[6] OR "DB_GENERAL".Estados[8]) AND NOT "DB_INC_GENERAL".Alarma_On THEN
       "MC_MoveRelative_DB"(Axis := "Eje_X",   // MC_MoveRelative
                            Execute := true,
                            Distance := "Cuentas_Matematicas1_DB".MovYNeg,
                            Done => #DoneY);
   END_IF;
END_REGION

REGION Network 49: Movimiento +2X
   IF "DB_GENERAL".Estados[14] AND NOT "DB_INC_GENERAL".Alarma_On THEN
       "MC_MoveRelative_DB"(Axis := "Eje_X",   // MC_MoveRelative
                            Execute := true,
                            Distance := "Cuentas_Matematicas1_DB".Mov2X,
                            Done => #Done2X);
   END_IF;
END_REGION

REGION Network 50: Movimiento -2X
   IF "DB_GENERAL".Estados[16] AND NOT "DB_INC_GENERAL".Alarma_On THEN
       "MC_MoveRelative_DB"(Axis := "Eje_X",   // MC_MoveRelative
                            Execute := true,
                            Distance := "Cuentas_Matematicas1_DB".Mov2XNeg,
                            Done => #Done2X);
   END_IF;
END_REGION

REGION Network 51: Avance inverter
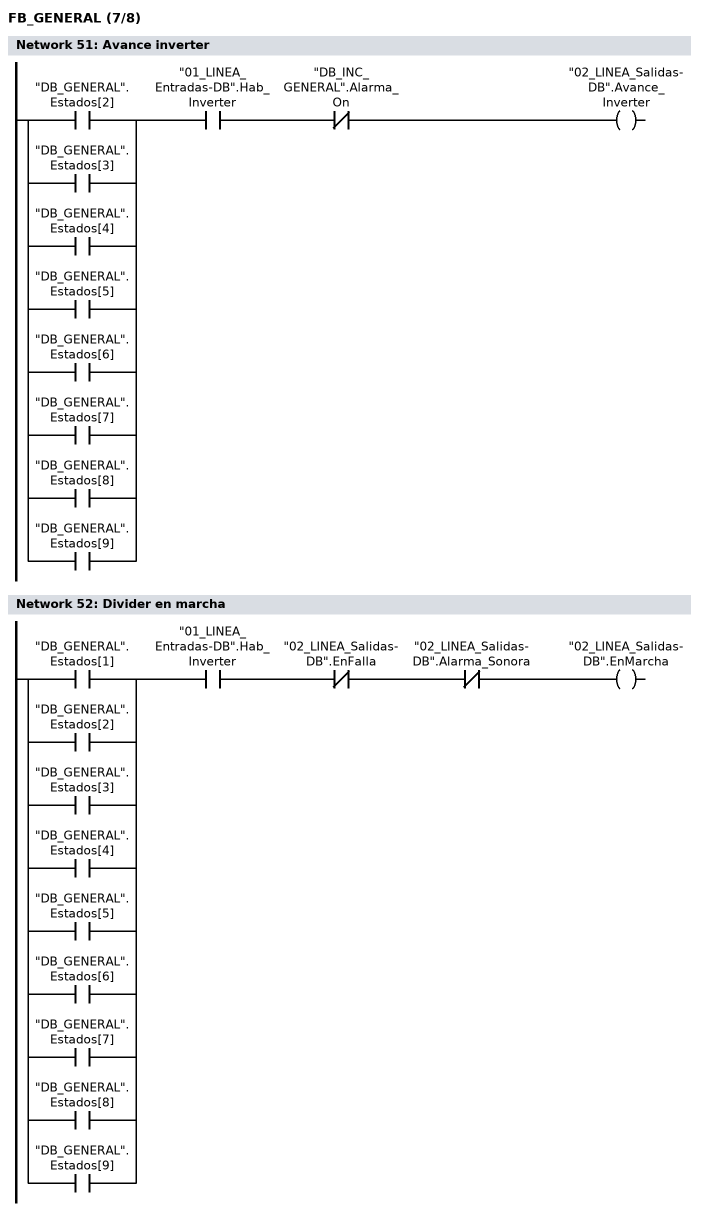
   RUNG wire#powerrail
      Contact( "DB_GENERAL".Estados[2] )
      wire#w1
      Contact( "01_LINEA_Entradas-DB".Hab_Inverter )
      I_Contact( "DB_INC_GENERAL".Alarma_On )
      Coil( "02_LINEA_Salidas-DB".Avance_Inverter )
   END_RUNG
   RUNG wire#powerrail
      Contact( "DB_GENERAL".Estados[3] )
   END_RUNG wire#w1
   RUNG wire#powerrail
      Contact( "DB_GENERAL".Estados[4] )
   END_RUNG wire#w1
   RUNG wire#powerrail
      Contact( "DB_GENERAL".Estados[5] )
   END_RUNG wire#w1
   RUNG wire#powerrail
      Contact( "DB_GENERAL".Estados[6] )
   END_RUNG wire#w1
   RUNG wire#powerrail
      Contact( "DB_GENERAL".Estados[7] )
   END_RUNG wire#w1
   RUNG wire#powerrail
      Contact( "DB_GENERAL".Estados[8] )
   END_RUNG wire#w1
   RUNG wire#powerrail
      Contact( "DB_GENERAL".Estados[9] )
   END_RUNG wire#w1
   // the same network as SCL:
   "02_LINEA_Salidas-DB".Avance_Inverter := ("DB_GENERAL".Estados[2] OR "DB_GENERAL".Estados[3] OR "DB_GENERAL".Estados[4] OR "DB_GENERAL".Estados[5] OR "DB_GENERAL".Estados[6] OR "DB_GENERAL".Estados[7] OR "DB_GENERAL".Estados[8] OR "DB_GENERAL".Estados[9]) AND "01_LINEA_Entradas-DB".Hab_Inverter AND NOT "DB_INC_GENERAL".Alarma_On;
END_REGION

REGION Network 52: Divider en marcha
   RUNG wire#powerrail
      Contact( "DB_GENERAL".Estados[1] )
      wire#w1
      Contact( "01_LINEA_Entradas-DB".Hab_Inverter )
      I_Contact( "02_LINEA_Salidas-DB".EnFalla )
      I_Contact( "02_LINEA_Salidas-DB".Alarma_Sonora )
      Coil( "02_LINEA_Salidas-DB".EnMarcha )
   END_RUNG
   RUNG wire#powerrail
      Contact( "DB_GENERAL".Estados[2] )
   END_RUNG wire#w1
   RUNG wire#powerrail
      Contact( "DB_GENERAL".Estados[3] )
   END_RUNG wire#w1
   RUNG wire#powerrail
      Contact( "DB_GENERAL".Estados[4] )
   END_RUNG wire#w1
   RUNG wire#powerrail
      Contact( "DB_GENERAL".Estados[5] )
   END_RUNG wire#w1
   RUNG wire#powerrail
      Contact( "DB_GENERAL".Estados[6] )
   END_RUNG wire#w1
   RUNG wire#powerrail
      Contact( "DB_GENERAL".Estados[7] )
   END_RUNG wire#w1
   RUNG wire#powerrail
      Contact( "DB_GENERAL".Estados[8] )
   END_RUNG wire#w1
   RUNG wire#powerrail
      Contact( "DB_GENERAL".Estados[9] )
   END_RUNG wire#w1
   // the same network as SCL:
   "02_LINEA_Salidas-DB".EnMarcha := ("DB_GENERAL".Estados[1] OR "DB_GENERAL".Estados[2] OR "DB_GENERAL".Estados[3] OR "DB_GENERAL".Estados[4] OR "DB_GENERAL".Estados[5] OR "DB_GENERAL".Estados[6] OR "DB_GENERAL".Estados[7] OR "DB_GENERAL".Estados[8] OR "DB_GENERAL".Estados[9]) AND "01_LINEA_Entradas-DB".Hab_Inverter AND NOT "02_LINEA_Salidas-DB".EnFalla AND NOT "02_LINEA_Salidas-DB".Alarma_Sonora;
END_REGION

REGION Network 53: Testigo de divider en marcha
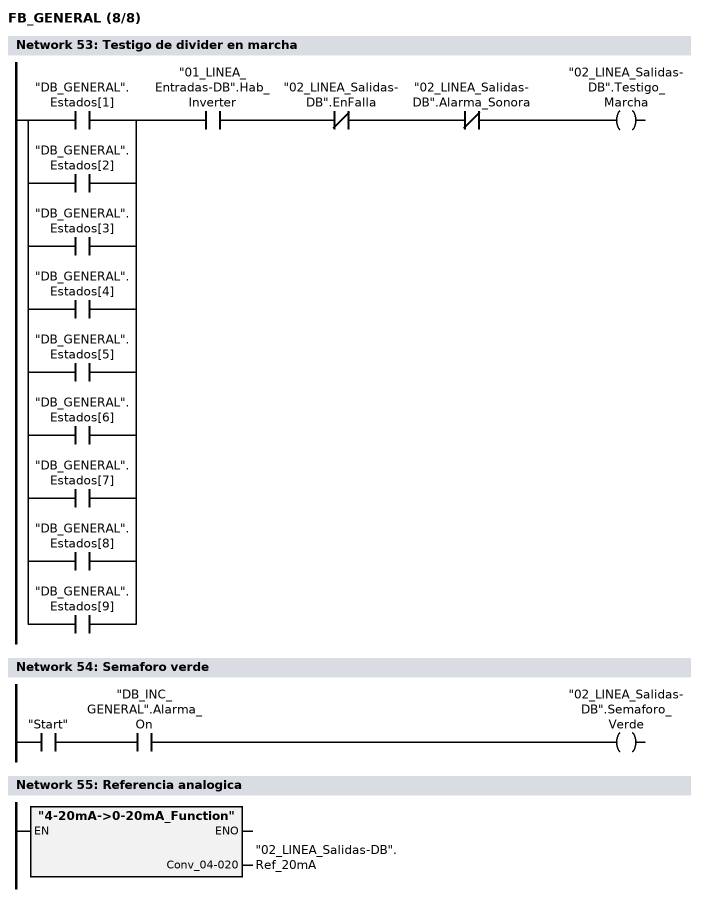
   RUNG wire#powerrail
      Contact( "DB_GENERAL".Estados[1] )
      wire#w1
      Contact( "01_LINEA_Entradas-DB".Hab_Inverter )
      I_Contact( "02_LINEA_Salidas-DB".EnFalla )
      I_Contact( "02_LINEA_Salidas-DB".Alarma_Sonora )
      Coil( "02_LINEA_Salidas-DB".Testigo_Marcha )
   END_RUNG
   RUNG wire#powerrail
      Contact( "DB_GENERAL".Estados[2] )
   END_RUNG wire#w1
   RUNG wire#powerrail
      Contact( "DB_GENERAL".Estados[3] )
   END_RUNG wire#w1
   RUNG wire#powerrail
      Contact( "DB_GENERAL".Estados[4] )
   END_RUNG wire#w1
   RUNG wire#powerrail
      Contact( "DB_GENERAL".Estados[5] )
   END_RUNG wire#w1
   RUNG wire#powerrail
      Contact( "DB_GENERAL".Estados[6] )
   END_RUNG wire#w1
   RUNG wire#powerrail
      Contact( "DB_GENERAL".Estados[7] )
   END_RUNG wire#w1
   RUNG wire#powerrail
      Contact( "DB_GENERAL".Estados[8] )
   END_RUNG wire#w1
   RUNG wire#powerrail
      Contact( "DB_GENERAL".Estados[9] )
   END_RUNG wire#w1
   // the same network as SCL:
   "02_LINEA_Salidas-DB".Testigo_Marcha := ("DB_GENERAL".Estados[1] OR "DB_GENERAL".Estados[2] OR "DB_GENERAL".Estados[3] OR "DB_GENERAL".Estados[4] OR "DB_GENERAL".Estados[5] OR "DB_GENERAL".Estados[6] OR "DB_GENERAL".Estados[7] OR "DB_GENERAL".Estados[8] OR "DB_GENERAL".Estados[9]) AND "01_LINEA_Entradas-DB".Hab_Inverter AND NOT "02_LINEA_Salidas-DB".EnFalla AND NOT "02_LINEA_Salidas-DB".Alarma_Sonora;
END_REGION

REGION Network 54: Semaforo verde
   RUNG wire#powerrail
      Contact( "Start" )
      Contact( "DB_INC_GENERAL".Alarma_On )
      Coil( "02_LINEA_Salidas-DB".Semaforo_Verde )
   END_RUNG
   // the same network as SCL:
   "02_LINEA_Salidas-DB".Semaforo_Verde := "Start" AND "DB_INC_GENERAL".Alarma_On;
END_REGION

REGION Network 55: Referencia analogica
   RUNG wire#powerrail
      "4-20mA->0-20mA_Function"("Conv_04-020" => "02_LINEA_Salidas-DB".Ref_20mA)
   END_RUNG
   // the same network as SCL:
   "4-20mA->0-20mA_Function"("Conv_04-020" => "02_LINEA_Salidas-DB".Ref_20mA);
END_REGION
END_FUNCTION_BLOCK

FUNCTION "01_LINEA_Entradas" : Void   // FC1, LAD
TITLE = Bloque de entradas
{ S7_Optimized_Access := 'TRUE' }
VERSION : 0.1
BEGIN

REGION Network 1: Contador
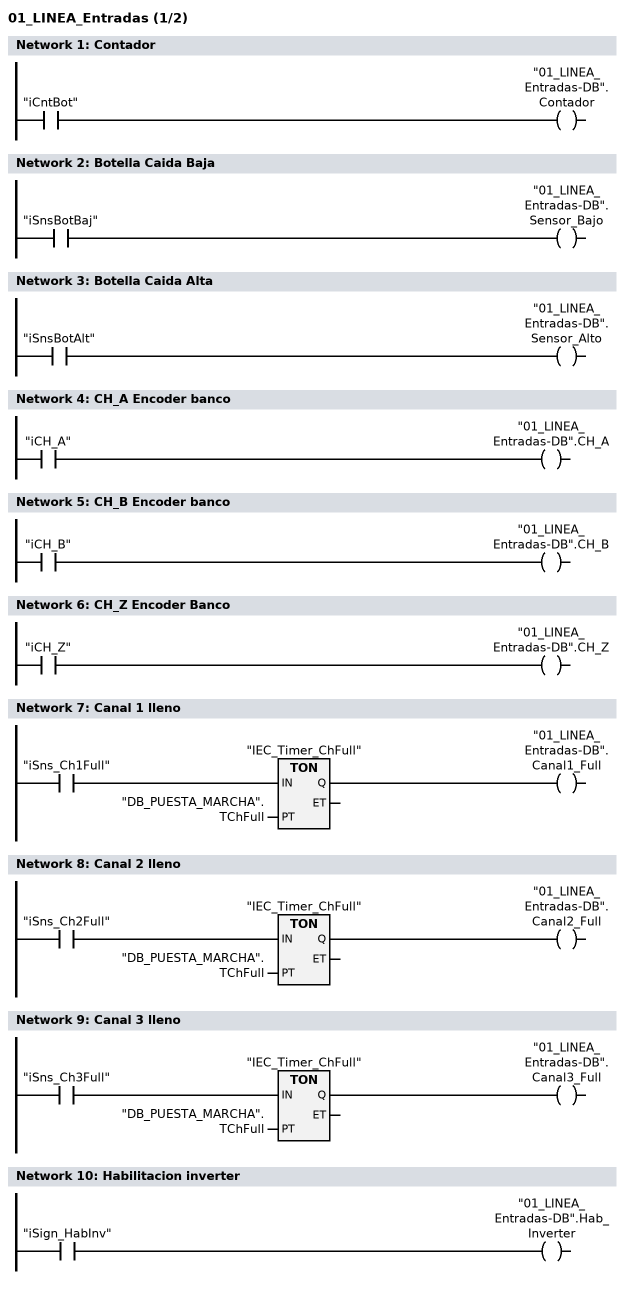
   RUNG wire#powerrail
      Contact( "iCntBot" )
      Coil( "01_LINEA_Entradas-DB".Contador )
   END_RUNG
   // the same network as SCL:
   "01_LINEA_Entradas-DB".Contador := "iCntBot";
END_REGION

REGION Network 2: Botella Caida Baja
   RUNG wire#powerrail
      Contact( "iSnsBotBaj" )
      Coil( "01_LINEA_Entradas-DB".Sensor_Bajo )
   END_RUNG
   // the same network as SCL:
   "01_LINEA_Entradas-DB".Sensor_Bajo := "iSnsBotBaj";
END_REGION

REGION Network 3: Botella Caida Alta
   RUNG wire#powerrail
      Contact( "iSnsBotAlt" )
      Coil( "01_LINEA_Entradas-DB".Sensor_Alto )
   END_RUNG
   // the same network as SCL:
   "01_LINEA_Entradas-DB".Sensor_Alto := "iSnsBotAlt";
END_REGION

REGION Network 4: CH_A Encoder banco
   RUNG wire#powerrail
      Contact( "iCH_A" )
      Coil( "01_LINEA_Entradas-DB".CH_A )
   END_RUNG
   // the same network as SCL:
   "01_LINEA_Entradas-DB".CH_A := "iCH_A";
END_REGION

REGION Network 5: CH_B Encoder banco
   RUNG wire#powerrail
      Contact( "iCH_B" )
      Coil( "01_LINEA_Entradas-DB".CH_B )
   END_RUNG
   // the same network as SCL:
   "01_LINEA_Entradas-DB".CH_B := "iCH_B";
END_REGION

REGION Network 6: CH_Z Encoder Banco
   RUNG wire#powerrail
      Contact( "iCH_Z" )
      Coil( "01_LINEA_Entradas-DB".CH_Z )
   END_RUNG
   // the same network as SCL:
   "01_LINEA_Entradas-DB".CH_Z := "iCH_Z";
END_REGION

REGION Network 7: Canal 1 lleno
   "IEC_Timer_ChFull".TON(IN := "iSns_Ch1Full", PT := "DB_PUESTA_MARCHA".TChFull);
   "01_LINEA_Entradas-DB".Canal1_Full := "IEC_Timer_ChFull".Q;
END_REGION

REGION Network 8: Canal 2 lleno
   "IEC_Timer_ChFull".TON(IN := "iSns_Ch2Full", PT := "DB_PUESTA_MARCHA".TChFull);
   "01_LINEA_Entradas-DB".Canal2_Full := "IEC_Timer_ChFull".Q;
END_REGION

REGION Network 9: Canal 3 lleno
   "IEC_Timer_ChFull".TON(IN := "iSns_Ch3Full", PT := "DB_PUESTA_MARCHA".TChFull);
   "01_LINEA_Entradas-DB".Canal3_Full := "IEC_Timer_ChFull".Q;
END_REGION

REGION Network 10: Habilitacion inverter
   RUNG wire#powerrail
      Contact( "iSign_HabInv" )
      Coil( "01_LINEA_Entradas-DB".Hab_Inverter )
   END_RUNG
   // the same network as SCL:
   "01_LINEA_Entradas-DB".Hab_Inverter := "iSign_HabInv";
END_REGION

REGION Network 11: Pulsador de Marcha de la columna 11
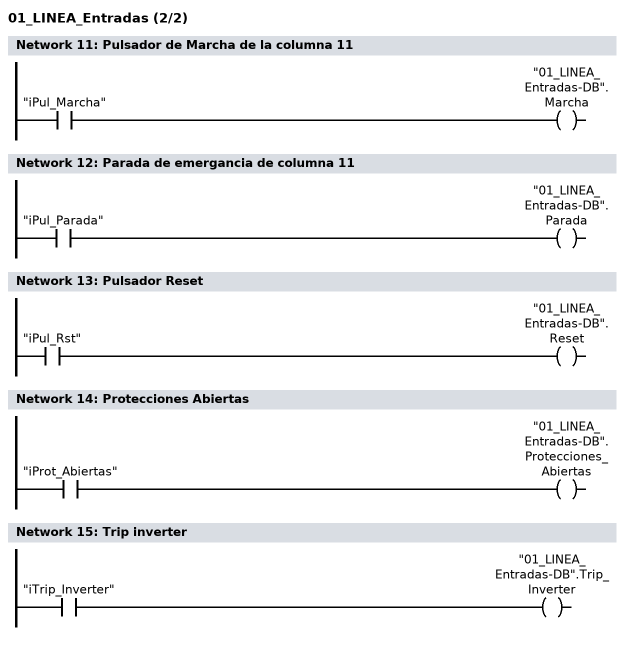
   RUNG wire#powerrail
      Contact( "iPul_Marcha" )
      Coil( "01_LINEA_Entradas-DB".Marcha )
   END_RUNG
   // the same network as SCL:
   "01_LINEA_Entradas-DB".Marcha := "iPul_Marcha";
END_REGION

REGION Network 12: Parada de emergancia de columna 11
   RUNG wire#powerrail
      Contact( "iPul_Parada" )
      Coil( "01_LINEA_Entradas-DB".Parada )
   END_RUNG
   // the same network as SCL:
   "01_LINEA_Entradas-DB".Parada := "iPul_Parada";
END_REGION

REGION Network 13: Pulsador Reset
   RUNG wire#powerrail
      Contact( "iPul_Rst" )
      Coil( "01_LINEA_Entradas-DB".Reset )
   END_RUNG
   // the same network as SCL:
   "01_LINEA_Entradas-DB".Reset := "iPul_Rst";
END_REGION

REGION Network 14: Protecciones Abiertas
   RUNG wire#powerrail
      Contact( "iProt_Abiertas" )
      Coil( "01_LINEA_Entradas-DB".Protecciones_Abiertas )
   END_RUNG
   // the same network as SCL:
   "01_LINEA_Entradas-DB".Protecciones_Abiertas := "iProt_Abiertas";
END_REGION

REGION Network 15: Trip inverter
   RUNG wire#powerrail
      Contact( "iTrip_Inverter" )
      Coil( "01_LINEA_Entradas-DB".Trip_Inverter )
   END_RUNG
   // the same network as SCL:
   "01_LINEA_Entradas-DB".Trip_Inverter := "iTrip_Inverter";
END_REGION
END_FUNCTION

FUNCTION "02_LINEA_Salidas" : Void   // FC2, LAD
{ S7_Optimized_Access := 'TRUE' }
VERSION : 0.1
BEGIN

REGION Network 1: Alarma Sonora
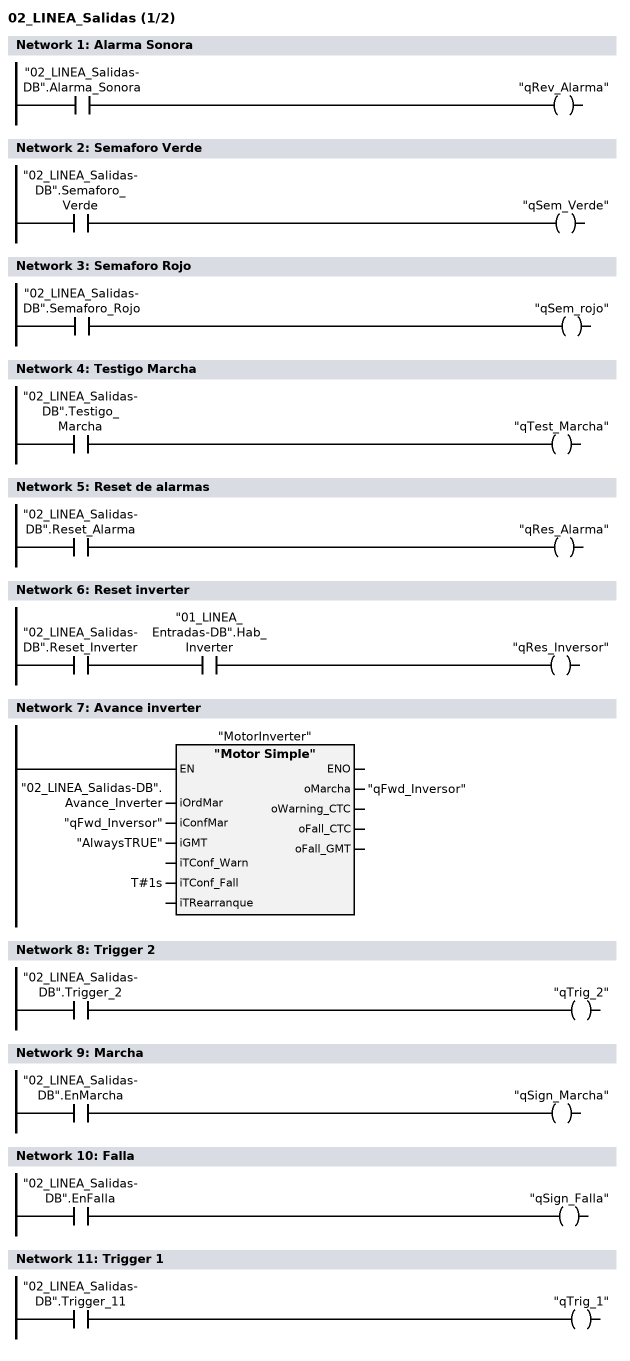
   RUNG wire#powerrail
      Contact( "02_LINEA_Salidas-DB".Alarma_Sonora )
      Coil( "qRev_Alarma" )
   END_RUNG
   // the same network as SCL:
   "qRev_Alarma" := "02_LINEA_Salidas-DB".Alarma_Sonora;
END_REGION

REGION Network 2: Semaforo Verde
   RUNG wire#powerrail
      Contact( "02_LINEA_Salidas-DB".Semaforo_Verde )
      Coil( "qSem_Verde" )
   END_RUNG
   // the same network as SCL:
   "qSem_Verde" := "02_LINEA_Salidas-DB".Semaforo_Verde;
END_REGION

REGION Network 3: Semaforo Rojo
   RUNG wire#powerrail
      Contact( "02_LINEA_Salidas-DB".Semaforo_Rojo )
      Coil( "qSem_rojo" )
   END_RUNG
   // the same network as SCL:
   "qSem_rojo" := "02_LINEA_Salidas-DB".Semaforo_Rojo;
END_REGION

REGION Network 4: Testigo Marcha
   RUNG wire#powerrail
      Contact( "02_LINEA_Salidas-DB".Testigo_Marcha )
      Coil( "qTest_Marcha" )
   END_RUNG
   // the same network as SCL:
   "qTest_Marcha" := "02_LINEA_Salidas-DB".Testigo_Marcha;
END_REGION

REGION Network 5: Reset de alarmas
   RUNG wire#powerrail
      Contact( "02_LINEA_Salidas-DB".Reset_Alarma )
      Coil( "qRes_Alarma" )
   END_RUNG
   // the same network as SCL:
   "qRes_Alarma" := "02_LINEA_Salidas-DB".Reset_Alarma;
END_REGION

REGION Network 6: Reset inverter
   RUNG wire#powerrail
      Contact( "02_LINEA_Salidas-DB".Reset_Inverter )
      Contact( "01_LINEA_Entradas-DB".Hab_Inverter )
      Coil( "qRes_Inversor" )
   END_RUNG
   // the same network as SCL:
   "qRes_Inversor" := "02_LINEA_Salidas-DB".Reset_Inverter AND "01_LINEA_Entradas-DB".Hab_Inverter;
END_REGION

REGION Network 7: Avance inverter
   RUNG wire#powerrail
      "MotorInverter"(iOrdMar := "02_LINEA_Salidas-DB".Avance_Inverter, iConfMar := "qFwd_Inversor", iGMT := "AlwaysTRUE", iTConf_Warn :=, iTConf_Fall := T#1s, iTRearranque :=, oMarcha => "qFwd_Inversor", oWarning_CTC =>, oFall_CTC =>, oFall_GMT =>)
   END_RUNG
   // the same network as SCL:
   "MotorInverter"(iOrdMar := "02_LINEA_Salidas-DB".Avance_Inverter,   // "Motor Simple"
                   iConfMar := "qFwd_Inversor",
                   iGMT := "AlwaysTRUE",
                   iTConf_Fall := T#1s,
                   oMarcha => "qFwd_Inversor");
END_REGION

REGION Network 8: Trigger 2
   RUNG wire#powerrail
      Contact( "02_LINEA_Salidas-DB".Trigger_2 )
      Coil( "qTrig_2" )
   END_RUNG
   // the same network as SCL:
   "qTrig_2" := "02_LINEA_Salidas-DB".Trigger_2;
END_REGION

REGION Network 9: Marcha
   RUNG wire#powerrail
      Contact( "02_LINEA_Salidas-DB".EnMarcha )
      Coil( "qSign_Marcha" )
   END_RUNG
   // the same network as SCL:
   "qSign_Marcha" := "02_LINEA_Salidas-DB".EnMarcha;
END_REGION

REGION Network 10: Falla
   RUNG wire#powerrail
      Contact( "02_LINEA_Salidas-DB".EnFalla )
      Coil( "qSign_Falla" )
   END_RUNG
   // the same network as SCL:
   "qSign_Falla" := "02_LINEA_Salidas-DB".EnFalla;
END_REGION

REGION Network 11: Trigger 1
   RUNG wire#powerrail
      Contact( "02_LINEA_Salidas-DB".Trigger_11 )
      Coil( "qTrig_1" )
   END_RUNG
   // the same network as SCL:
   "qTrig_1" := "02_LINEA_Salidas-DB".Trigger_11;
END_REGION

REGION Network 12: Trigger 22
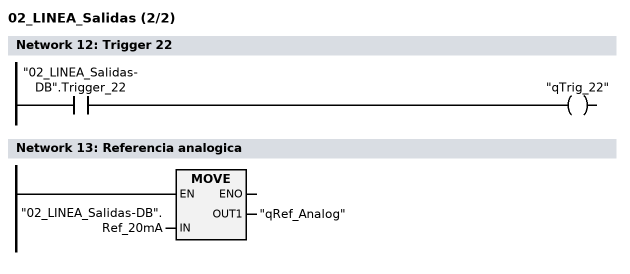
   RUNG wire#powerrail
      Contact( "02_LINEA_Salidas-DB".Trigger_22 )
      Coil( "qTrig_22" )
   END_RUNG
   // the same network as SCL:
   "qTrig_22" := "02_LINEA_Salidas-DB".Trigger_22;
END_REGION

REGION Network 13: Referencia analogica
   RUNG wire#powerrail
      Move(in := "02_LINEA_Salidas-DB".Ref_20mA, out1 => "qRef_Analog")
   END_RUNG
   // the same network as SCL:
   "qRef_Analog" := "02_LINEA_Salidas-DB".Ref_20mA;
END_REGION
END_FUNCTION

FUNCTION "4-20mA->0-20mA_Function" : Void   // FC3, LAD
TITLE = Conversion 4-20 -> 0-20 Canal 1
{ S7_Optimized_Access := 'TRUE' }
VERSION : 0.1
   VAR_OUTPUT
      "Conv_04-020" : Int;
   END_VAR
   VAR_TEMP
      Input_Analog1 : Real;
      Temp_Analog1 : Real;
      Input_Analog2 : Real;
      Temp_Analog2 : Real;
   END_VAR
BEGIN

REGION Network 1
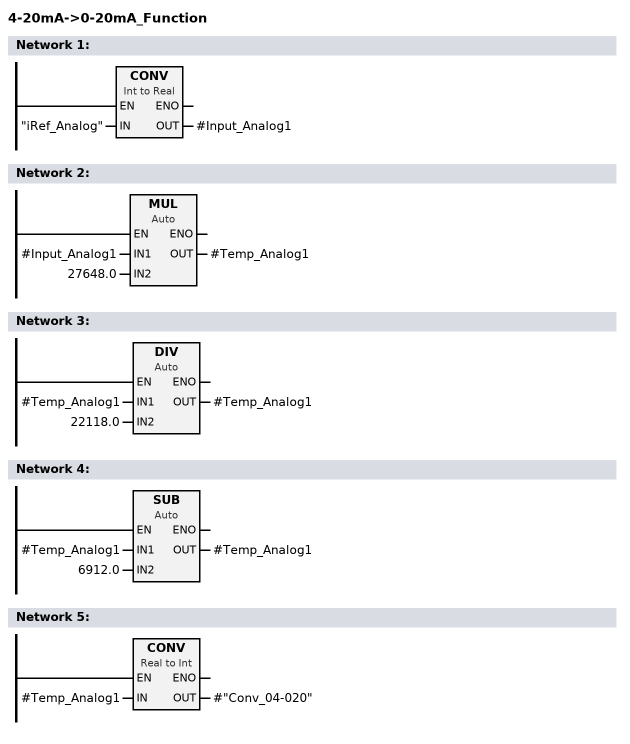
   RUNG wire#powerrail
      { S7_Templates := "[SrcType := Int, DestType := Real]" } Convert(in := "iRef_Analog", out => #Input_Analog1)
   END_RUNG
   // the same network as SCL:
   #Input_Analog1 := INT_TO_REAL("iRef_Analog");
END_REGION

REGION Network 2
   RUNG wire#powerrail
      Mul(in1 := #Input_Analog1, in2 := 27648.0, out => #Temp_Analog1)
   END_RUNG
   // the same network as SCL:
   #Temp_Analog1 := #Input_Analog1 * 27648.0;
END_REGION

REGION Network 3
   RUNG wire#powerrail
      Div(in1 := #Temp_Analog1, in2 := 22118.0, out => #Temp_Analog1)
   END_RUNG
   // the same network as SCL:
   #Temp_Analog1 := #Temp_Analog1 / 22118.0;
END_REGION

REGION Network 4
   RUNG wire#powerrail
      Sub(in1 := #Temp_Analog1, in2 := 6912.0, out => #Temp_Analog1)
   END_RUNG
   // the same network as SCL:
   #Temp_Analog1 := #Temp_Analog1 - 6912.0;
END_REGION

REGION Network 5
   RUNG wire#powerrail
      { S7_Templates := "[SrcType := Real, DestType := Int]" } Convert(in := #Temp_Analog1, out => #"Conv_04-020")
   END_RUNG
   // the same network as SCL:
   #"Conv_04-020" := REAL_TO_INT(#Temp_Analog1);
END_REGION
END_FUNCTION

ORGANIZATION_BLOCK "Main"   // OB1, LAD, ProgramCycle
TITLE = "Main Program Sweep (Cycle)"
{ S7_Optimized_Access := 'TRUE' }
VERSION : 0.1
   VAR_INPUT
      Initial_Call : Bool;   // Initial call of this OB
      Remanence : Bool;   // =True, if remanent data are available
   END_VAR
BEGIN

REGION Network 1
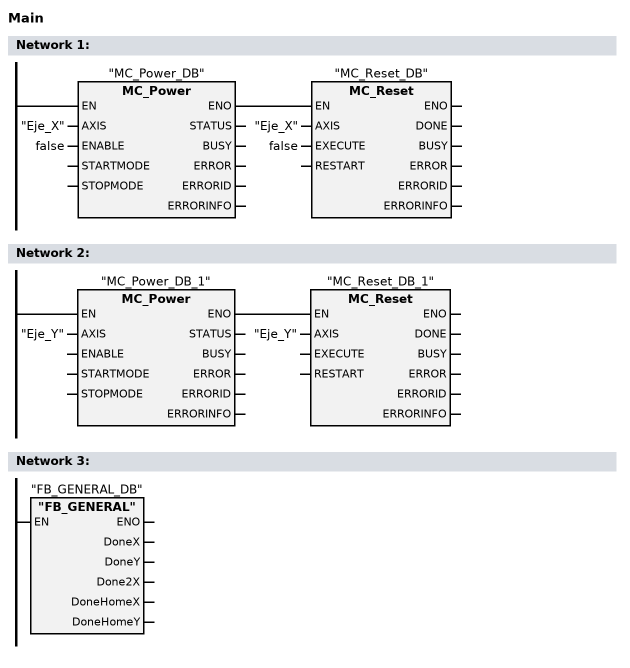
   // ENO of a box is taken as its EN; it also drops when the box reports an error
   "MC_Power_DB"(Axis := "Eje_X", Enable := false);   // MC_Power
   "MC_Reset_DB"(Axis := "Eje_X", Execute := false);   // MC_Reset
END_REGION

REGION Network 2
   // ENO of a box is taken as its EN; it also drops when the box reports an error
   "MC_Power_DB_1"(Axis := "Eje_Y");   // MC_Power
   "MC_Reset_DB_1"(Axis := "Eje_Y");   // MC_Reset
END_REGION

REGION Network 3
   RUNG wire#powerrail
      "FB_GENERAL_DB"(DoneX =>, DoneY =>, Done2X =>, DoneHomeX =>, DoneHomeY =>)
   END_RUNG
   // the same network as SCL:
   "FB_GENERAL_DB"();   // "FB_GENERAL"
END_REGION
END_ORGANIZATION_BLOCK

// folder: ESTANDAR

FUNCTION_BLOCK "Motor M&CM"   // FB2, LAD
TITLE = Motor Marcha & Contra-Marcha
{ S7_Optimized_Access := 'TRUE' }
VERSION : 0.1
   VAR_INPUT
      iOrdMar_Dir : Bool;
      iOrdMar_Rev : Bool;
      iConfMar_Dir : Bool;
      iConfMar_Rev : Bool;
      iGMT : Bool;
      iTConf_Warn : Time;
      iTConf_Fall : Time;
      iTRearranque : Time;
   END_VAR
   VAR_OUTPUT
      oMar_Dir : Bool;
      oMar_Rev : Bool;
      oWarning_CTC_Dir : Bool;
      oWarning_CTC_Rev : Bool;
      oFall_CTC_Dir : Bool;
      oFall_CTC_Rev : Bool;
      oFall_GMT : Bool;
   END_VAR
   VAR
      IEC_Timer_0_Instance : IEC_TIMER;
      IEC_Timer_0_Instance_1 : IEC_TIMER;
      IEC_Timer_0_Instance_2 : IEC_TIMER;
      IEC_Timer_0_Instance_3 : IEC_TIMER;
      IEC_Timer_0_Instance_4 : IEC_TIMER;
      MarDir_Aux : Bool;
      MarRev_Aux : Bool;
   END_VAR
   VAR_TEMP
      Fall_GMT_Aux : Bool;
      Fall_CTC_Dir_Aux : Bool;
      Fall_CTC_Rev_Aux : Bool;
      Habil_Mov : Bool;
   END_VAR
   VAR_TEMP   // added for the SCL form of the ladder/FBD networks
      _w1 : Bool;
   END_VAR
BEGIN

REGION Network 1: Falla Guardamotor
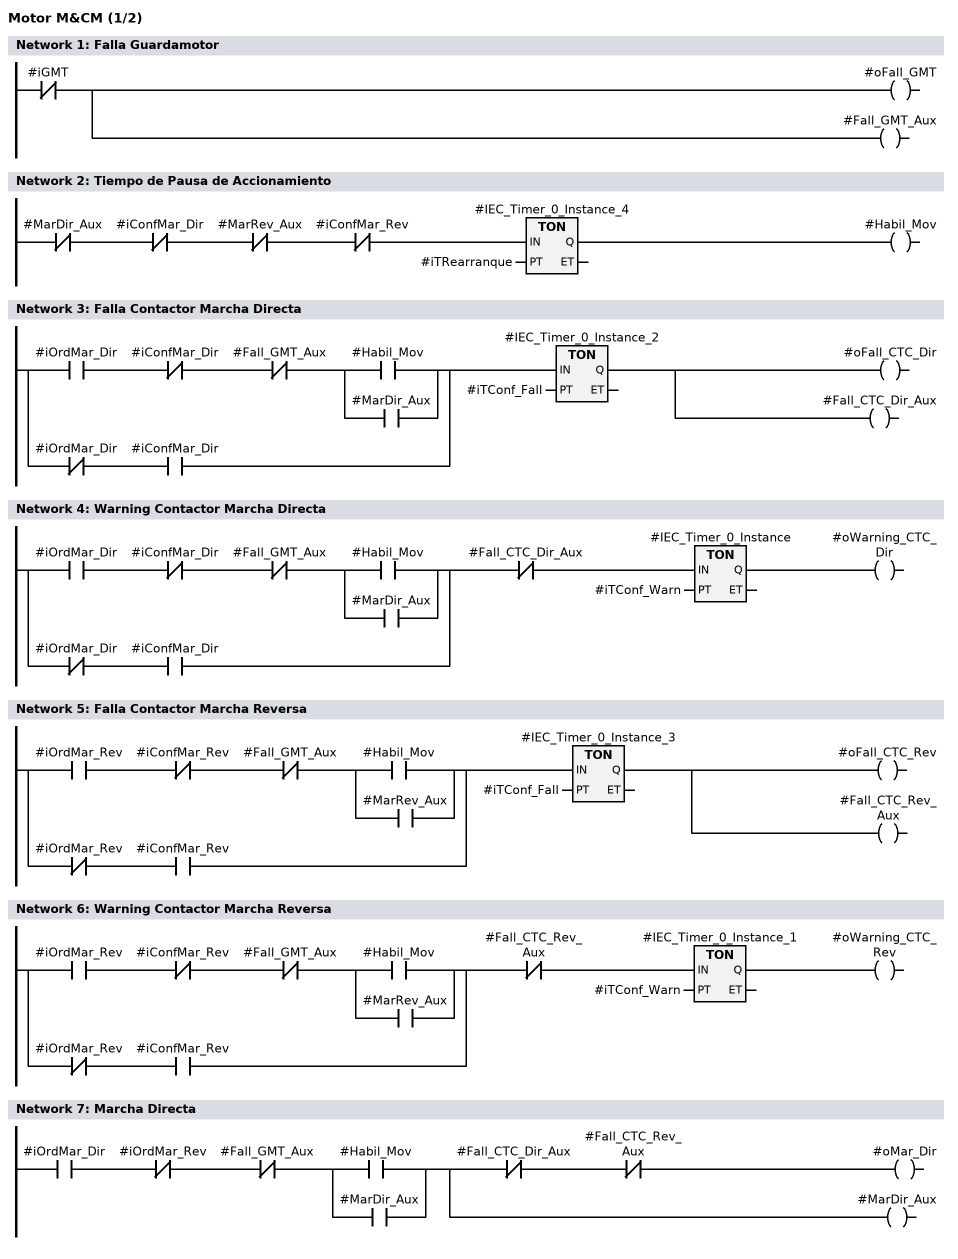
   RUNG wire#powerrail
      I_Contact( #iGMT )
      wire#w1
      Coil( #oFall_GMT )
   END_RUNG
   RUNG wire#w1
      Coil( #Fall_GMT_Aux )
   END_RUNG
   // the same network as SCL:
   #oFall_GMT := NOT #iGMT;
   #Fall_GMT_Aux := NOT #iGMT;
END_REGION

REGION Network 2: Tiempo de Pausa de Accionamiento
   #IEC_Timer_0_Instance_4.TON(IN := NOT #MarDir_Aux AND NOT #iConfMar_Dir AND NOT #MarRev_Aux AND NOT #iConfMar_Rev,
                           PT := #iTRearranque);
   #Habil_Mov := #IEC_Timer_0_Instance_4.Q;
END_REGION

REGION Network 3: Falla Contactor Marcha Directa
   #IEC_Timer_0_Instance_2.TON(IN := (#iOrdMar_Dir AND NOT #iConfMar_Dir AND NOT #Fall_GMT_Aux AND (#Habil_Mov OR #MarDir_Aux)) OR (NOT #iOrdMar_Dir AND #iConfMar_Dir),
                           PT := #iTConf_Fall);
   #oFall_CTC_Dir := #IEC_Timer_0_Instance_2.Q;
   #Fall_CTC_Dir_Aux := #IEC_Timer_0_Instance_2.Q;
END_REGION

REGION Network 4: Warning Contactor Marcha Directa
   #IEC_Timer_0_Instance.TON(IN := ((#iOrdMar_Dir AND NOT #iConfMar_Dir AND NOT #Fall_GMT_Aux AND (#Habil_Mov OR #MarDir_Aux)) OR (NOT #iOrdMar_Dir AND #iConfMar_Dir)) AND NOT #Fall_CTC_Dir_Aux,
                           PT := #iTConf_Warn);
   #oWarning_CTC_Dir := #IEC_Timer_0_Instance.Q;
END_REGION

REGION Network 5: Falla Contactor Marcha Reversa
   #IEC_Timer_0_Instance_3.TON(IN := (#iOrdMar_Rev AND NOT #iConfMar_Rev AND NOT #Fall_GMT_Aux AND (#Habil_Mov OR #MarRev_Aux)) OR (NOT #iOrdMar_Rev AND #iConfMar_Rev),
                           PT := #iTConf_Fall);
   #oFall_CTC_Rev := #IEC_Timer_0_Instance_3.Q;
   #Fall_CTC_Rev_Aux := #IEC_Timer_0_Instance_3.Q;
END_REGION

REGION Network 6: Warning Contactor Marcha Reversa
   #IEC_Timer_0_Instance_1.TON(IN := ((#iOrdMar_Rev AND NOT #iConfMar_Rev AND NOT #Fall_GMT_Aux AND (#Habil_Mov OR #MarRev_Aux)) OR (NOT #iOrdMar_Rev AND #iConfMar_Rev)) AND NOT #Fall_CTC_Rev_Aux,
                           PT := #iTConf_Warn);
   #oWarning_CTC_Rev := #IEC_Timer_0_Instance_1.Q;
END_REGION

REGION Network 7: Marcha Directa
   RUNG wire#powerrail
      Contact( #iOrdMar_Dir )
      I_Contact( #iOrdMar_Rev )
      I_Contact( #Fall_GMT_Aux )
      wire#w1
      Contact( #Habil_Mov )
      wire#w2
      I_Contact( #Fall_CTC_Dir_Aux )
      I_Contact( #Fall_CTC_Rev_Aux )
      Coil( #oMar_Dir )
   END_RUNG
   RUNG wire#w1
      Contact( #MarDir_Aux )
   END_RUNG wire#w2
   RUNG wire#w2
      Coil( #MarDir_Aux )
   END_RUNG
   // the same network as SCL:
   #_w1 := #iOrdMar_Dir AND NOT #iOrdMar_Rev AND NOT #Fall_GMT_Aux AND (#Habil_Mov OR #MarDir_Aux);
   #oMar_Dir := #_w1 AND NOT #Fall_CTC_Dir_Aux AND NOT #Fall_CTC_Rev_Aux;
   #MarDir_Aux := #_w1;
END_REGION

REGION Network 8: Marcha Reversa
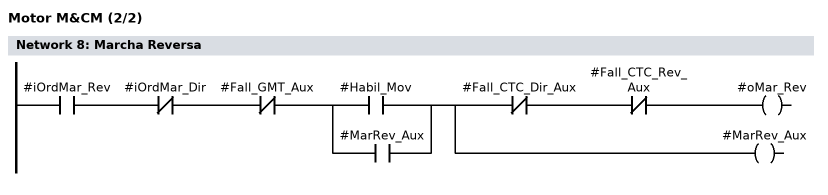
   RUNG wire#powerrail
      Contact( #iOrdMar_Rev )
      I_Contact( #iOrdMar_Dir )
      I_Contact( #Fall_GMT_Aux )
      wire#w1
      Contact( #Habil_Mov )
      wire#w2
      I_Contact( #Fall_CTC_Dir_Aux )
      I_Contact( #Fall_CTC_Rev_Aux )
      Coil( #oMar_Rev )
   END_RUNG
   RUNG wire#w1
      Contact( #MarRev_Aux )
   END_RUNG wire#w2
   RUNG wire#w2
      Coil( #MarRev_Aux )
   END_RUNG
   // the same network as SCL:
   #_w1 := #iOrdMar_Rev AND NOT #iOrdMar_Dir AND NOT #Fall_GMT_Aux AND (#Habil_Mov OR #MarRev_Aux);
   #oMar_Rev := #_w1 AND NOT #Fall_CTC_Dir_Aux AND NOT #Fall_CTC_Rev_Aux;
   #MarRev_Aux := #_w1;
END_REGION
END_FUNCTION_BLOCK

FUNCTION_BLOCK "FB_VAR_MOT"   // FB4, LAD
{ S7_Optimized_Access := 'FALSE' }
VERSION : 0.1
   VAR_INPUT
      "CMD Mar Dir" : Bool;   // Comando Marcha Directa
      "CMD Mar Rev" : Bool;   // Comando Marcha Reversa
      "HAB  Mar" : Bool;   // Habilita Marcha
      "SP Vel" : Real;   // Setpoint de Velocidad
      Reset : Bool;   // Comando resetear falla
      Fault : Bool;   // Indica variador en falla
      Ready : Bool;   // Indica variador Ready
      Ton_Freno : Time := T#400ms;
      Ton_Mar : Time := T#100ms;
      Tof_Freno : Time := T#100ms;
      Tof_Mar : Time := T#200ms;
   END_VAR
   VAR_OUTPUT
      Marcha : Bool;   // Orden de marcha a variador
      "Inv Giro" : Bool;   // Orden de invertir sentido de giro a variador
      "Reset Fault" : Bool;   // Reset Fault a variador
      Velocidad : Word;   // Referencia de Velocidad a variador
      Freno : Bool;   // Apertura de Freno
      Falla : Bool;   // Indica falla del variador
      Warning : Bool;   // Indica variador no Ready
   END_VAR
   VAR
      IEC_Timer_Freno : TON_TIME;
      IEC_Timer_Motor : TON_TIME;
      IEC_Timer_Reset : TOF_TIME;
      "_CMD Marcha Dir" : Bool;
      "_CMD Marcha Rev" : Bool;
      _CMD_AbrirFreno : Bool;
      IEC_Timer_0_Instance : TON_TIME;
      IEC_Timer_0_Instance_1 : TOF_TIME;
      IEC_Timer_0_Instance_2 : TOF_TIME;
      Ord_Marcha : Bool;
      Mem_Inv : Bool;
   END_VAR
   VAR_TEMP
      Vel_Real : Real;
      Vel_Int : Int;
      _Hab_Abrir_Freno : Bool;
      "Pre Marcha" : Bool;
      Aux : Bool;
      Freno_Aux : Bool;
   END_VAR
   VAR_TEMP   // added for the SCL form of the ladder/FBD networks
      _w1 : Bool;
      _w2 : Bool;
      _w3 : Bool;
   END_VAR
BEGIN

REGION Network 1: #Aux
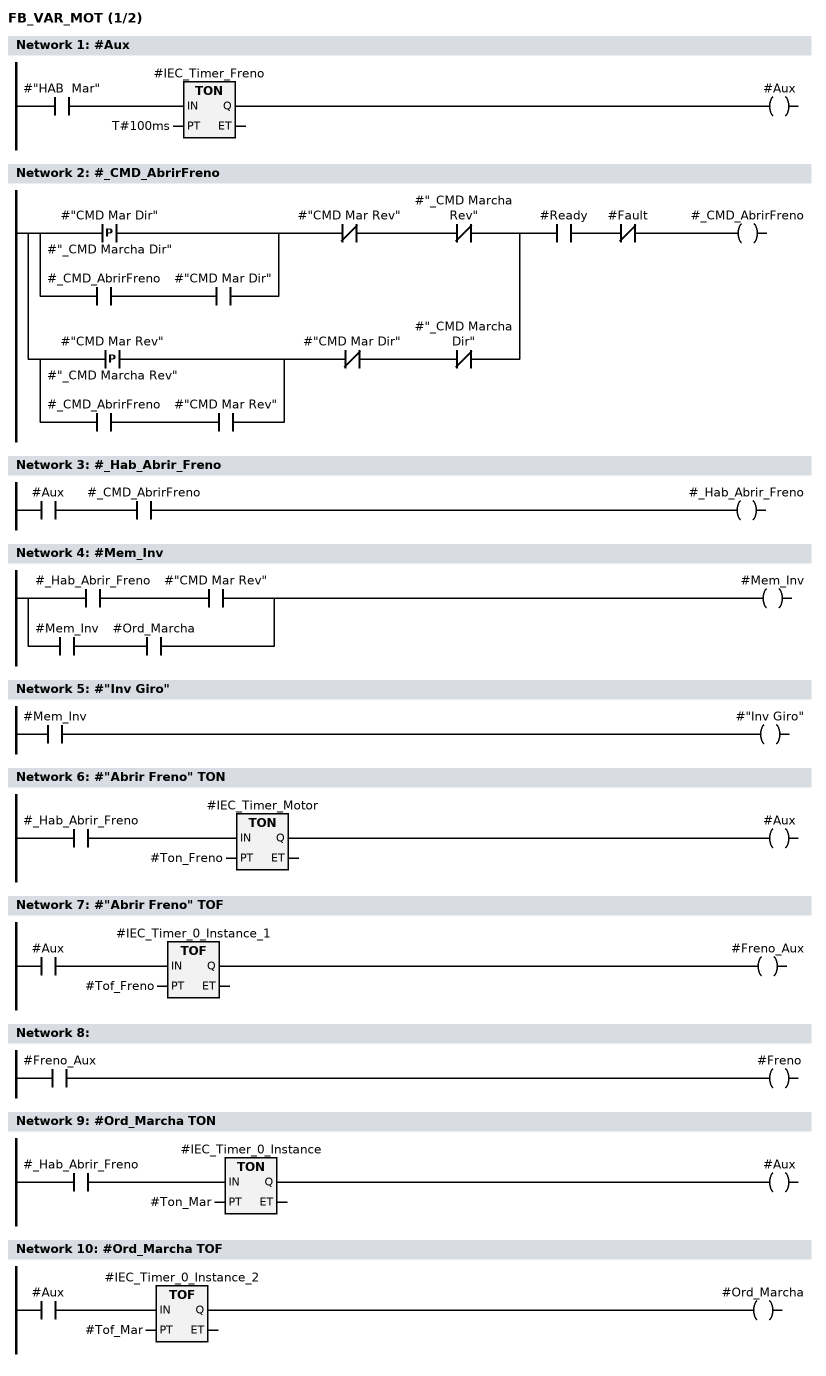
   #IEC_Timer_Freno(IN := #"HAB  Mar", PT := T#100ms);   // TON
   #Aux := #IEC_Timer_Freno.Q;
END_REGION

REGION Network 2: #_CMD_AbrirFreno
   RUNG wire#powerrail
      P_Contact(operand := #"CMD Mar Dir", bit := #"_CMD Marcha Dir")
      wire#w1
      I_Contact( #"CMD Mar Rev" )
      I_Contact( #"_CMD Marcha Rev" )
      wire#w2
      Contact( #Ready )
      I_Contact( #Fault )
      Coil( #_CMD_AbrirFreno )
   END_RUNG
   RUNG wire#powerrail
      Contact( #_CMD_AbrirFreno )
      Contact( #"CMD Mar Dir" )
   END_RUNG wire#w1
   RUNG wire#powerrail
      P_Contact(operand := #"CMD Mar Rev", bit := #"_CMD Marcha Rev")
      wire#w3
      I_Contact( #"CMD Mar Dir" )
      I_Contact( #"_CMD Marcha Dir" )
   END_RUNG wire#w2
   RUNG wire#powerrail
      Contact( #_CMD_AbrirFreno )
      Contact( #"CMD Mar Rev" )
   END_RUNG wire#w3
   // the same network as SCL:
   #_w1 := #"CMD Mar Dir" AND NOT #"_CMD Marcha Dir";   // rising edge of #"CMD Mar Dir"
   #"_CMD Marcha Dir" := #"CMD Mar Dir";
   #_w3 := (#_w1 OR (#_CMD_AbrirFreno AND #"CMD Mar Dir")) AND NOT #"CMD Mar Rev" AND NOT #"_CMD Marcha Rev";
   #_w2 := #"CMD Mar Rev" AND NOT #"_CMD Marcha Rev";   // rising edge of #"CMD Mar Rev"
   #"_CMD Marcha Rev" := #"CMD Mar Rev";
   #_CMD_AbrirFreno := (#_w3 OR ((#_w2 OR (#_CMD_AbrirFreno AND #"CMD Mar Rev")) AND NOT #"CMD Mar Dir" AND NOT #"_CMD Marcha Dir")) AND #Ready AND NOT #Fault;
END_REGION

REGION Network 3: #_Hab_Abrir_Freno
   RUNG wire#powerrail
      Contact( #Aux )
      Contact( #_CMD_AbrirFreno )
      Coil( #_Hab_Abrir_Freno )
   END_RUNG
   // the same network as SCL:
   #_Hab_Abrir_Freno := #Aux AND #_CMD_AbrirFreno;
END_REGION

REGION Network 4: #Mem_Inv
   RUNG wire#powerrail
      Contact( #_Hab_Abrir_Freno )
      Contact( #"CMD Mar Rev" )
      wire#w1
      Coil( #Mem_Inv )
   END_RUNG
   RUNG wire#powerrail
      Contact( #Mem_Inv )
      Contact( #Ord_Marcha )
   END_RUNG wire#w1
   // the same network as SCL:
   #Mem_Inv := (#_Hab_Abrir_Freno AND #"CMD Mar Rev") OR (#Mem_Inv AND #Ord_Marcha);
END_REGION

REGION Network 5: #"Inv Giro"
   RUNG wire#powerrail
      Contact( #Mem_Inv )
      Coil( #"Inv Giro" )
   END_RUNG
   // the same network as SCL:
   #"Inv Giro" := #Mem_Inv;
END_REGION

REGION Network 6: #"Abrir Freno" TON
   #IEC_Timer_Motor(IN := #_Hab_Abrir_Freno, PT := #Ton_Freno);   // TON
   #Aux := #IEC_Timer_Motor.Q;
END_REGION

REGION Network 7: #"Abrir Freno" TOF
   #IEC_Timer_0_Instance_1(IN := #Aux, PT := #Tof_Freno);   // TOF
   #Freno_Aux := #IEC_Timer_0_Instance_1.Q;
END_REGION

REGION Network 8
   RUNG wire#powerrail
      Contact( #Freno_Aux )
      Coil( #Freno )
   END_RUNG
   // the same network as SCL:
   #Freno := #Freno_Aux;
END_REGION

REGION Network 9: #Ord_Marcha TON
   #IEC_Timer_0_Instance(IN := #_Hab_Abrir_Freno, PT := #Ton_Mar);   // TON
   #Aux := #IEC_Timer_0_Instance.Q;
END_REGION

REGION Network 10: #Ord_Marcha TOF
   #IEC_Timer_0_Instance_2(IN := #Aux, PT := #Tof_Mar);   // TOF
   #Ord_Marcha := #IEC_Timer_0_Instance_2.Q;
END_REGION

REGION Network 11: #Marcha
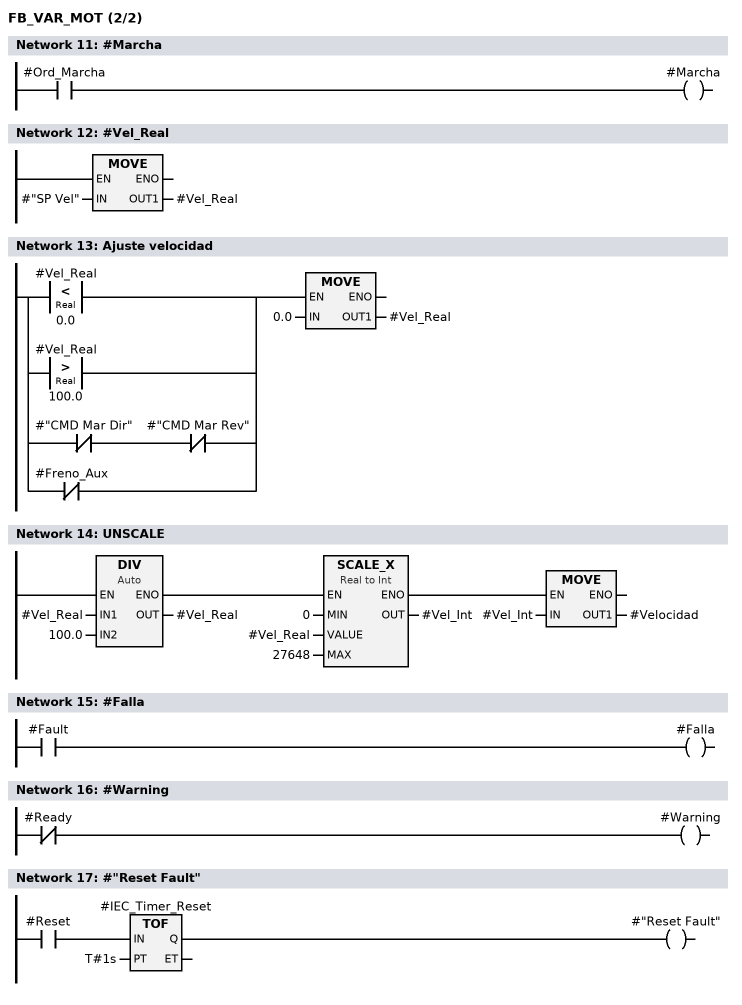
   RUNG wire#powerrail
      Contact( #Ord_Marcha )
      Coil( #Marcha )
   END_RUNG
   // the same network as SCL:
   #Marcha := #Ord_Marcha;
END_REGION

REGION Network 12: #Vel_Real
   RUNG wire#powerrail
      { S7_GenerateENO := "TRUE" } Move(in := #"SP Vel", out1 => #Vel_Real)
   END_RUNG
   // the same network as SCL:
   #Vel_Real := #"SP Vel";
END_REGION

REGION Network 13: Ajuste velocidad
   RUNG wire#powerrail
      { S7_Templates := "SrcType := Real" } LT_Contact(in1 := #Vel_Real, in2 := 0.0)
      wire#w1
      { S7_GenerateENO := "TRUE" } Move(in := 0.0, out1 => #Vel_Real)
   END_RUNG
   RUNG wire#powerrail
      { S7_Templates := "SrcType := Real" } GT_Contact(in1 := #Vel_Real, in2 := 100.0)
   END_RUNG wire#w1
   RUNG wire#powerrail
      I_Contact( #"CMD Mar Dir" )
      I_Contact( #"CMD Mar Rev" )
   END_RUNG wire#w1
   RUNG wire#powerrail
      I_Contact( #Freno_Aux )
   END_RUNG wire#w1
   // the same network as SCL:
   IF (#Vel_Real < 0.0) OR (#Vel_Real > 100.0) OR (NOT #"CMD Mar Dir" AND NOT #"CMD Mar Rev") OR NOT #Freno_Aux THEN
       #Vel_Real := 0.0;
   END_IF;
END_REGION

REGION Network 14: UNSCALE
   RUNG wire#powerrail
      Div(in1 := #Vel_Real, in2 := 100.0, out => #Vel_Real)
      { S7_Templates := "[SrcType := Real, DestType := Int]" } Scale(min := 0, value := #Vel_Real, max := 27648, out => #Vel_Int)
      { S7_GenerateENO := "TRUE" } Move(in := #Vel_Int, out1 => #Velocidad)
   END_RUNG
   // the same network as SCL:
   #Vel_Real := #Vel_Real / 100.0;
   #Vel_Int := SCALE_X(MIN := 0, VALUE := #Vel_Real, MAX := 27648);
   #Velocidad := #Vel_Int;
END_REGION

REGION Network 15: #Falla
   RUNG wire#powerrail
      Contact( #Fault )
      Coil( #Falla )
   END_RUNG
   // the same network as SCL:
   #Falla := #Fault;
END_REGION

REGION Network 16: #Warning
   RUNG wire#powerrail
      I_Contact( #Ready )
      Coil( #Warning )
   END_RUNG
   // the same network as SCL:
   #Warning := NOT #Ready;
END_REGION

REGION Network 17: #"Reset Fault"
   #IEC_Timer_Reset(IN := #Reset, PT := T#1s);   // TOF
   #"Reset Fault" := #IEC_Timer_Reset.Q;
END_REGION
END_FUNCTION_BLOCK

FUNCTION_BLOCK "Motor Simple"   // FB5, LAD
{ S7_Optimized_Access := 'TRUE' }
VERSION : 0.1
   VAR_INPUT
      iOrdMar : Bool;
      iConfMar : Bool;
      iGMT : Bool;
      iTConf_Warn : Time;
      iTConf_Fall : Time;
      iTRearranque : Time;
   END_VAR
   VAR_OUTPUT
      oMarcha : Bool;
      oWarning_CTC : Bool;
      oFall_CTC : Bool;
      oFall_GMT : Bool;
   END_VAR
   VAR
      IEC_Timer_0_Instance : IEC_TIMER;
      IEC_Timer_0_Instance_1 : IEC_TIMER;
      IEC_Timer_0_Instance_2 : IEC_TIMER;
      Mar_Aux : Bool;
   END_VAR
   VAR_TEMP
      Fall_GMT_Aux : Bool;
      Fall_CTC_Aux : Bool;
      Habil_Mov : Bool;
   END_VAR
BEGIN

REGION Network 1: Falla Guardamotor
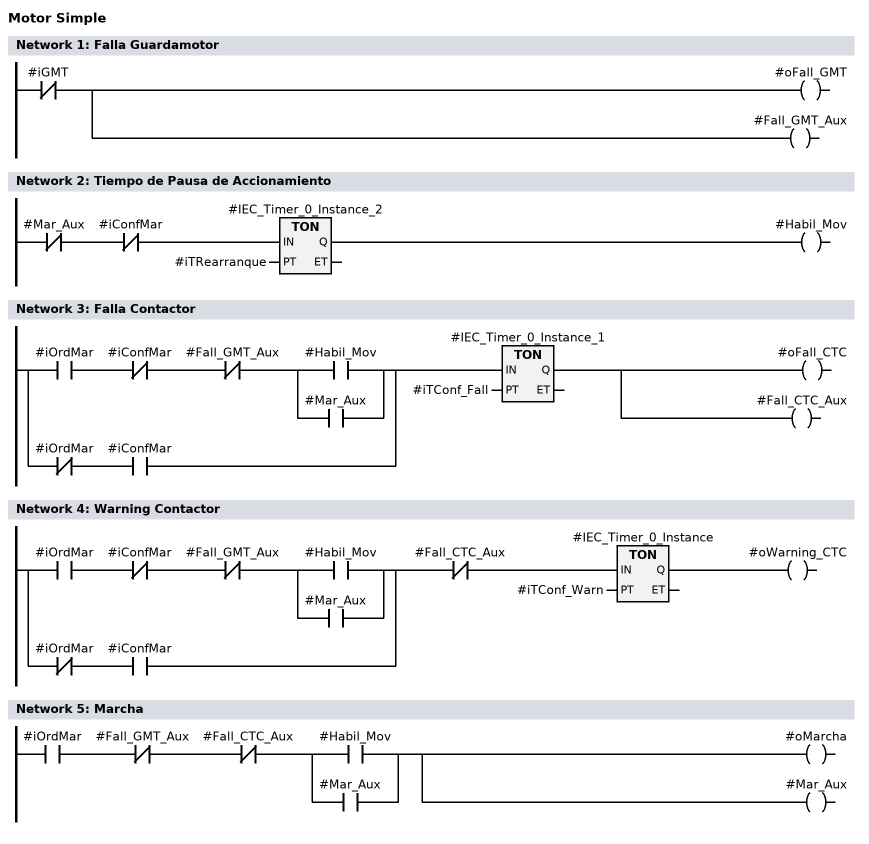
   RUNG wire#powerrail
      I_Contact( #iGMT )
      wire#w1
      Coil( #oFall_GMT )
   END_RUNG
   RUNG wire#w1
      Coil( #Fall_GMT_Aux )
   END_RUNG
   // the same network as SCL:
   #oFall_GMT := NOT #iGMT;
   #Fall_GMT_Aux := NOT #iGMT;
END_REGION

REGION Network 2: Tiempo de Pausa de Accionamiento
   #IEC_Timer_0_Instance_2.TON(IN := NOT #Mar_Aux AND NOT #iConfMar, PT := #iTRearranque);
   #Habil_Mov := #IEC_Timer_0_Instance_2.Q;
END_REGION

REGION Network 3: Falla Contactor
   #IEC_Timer_0_Instance_1.TON(IN := (#iOrdMar AND NOT #iConfMar AND NOT #Fall_GMT_Aux AND (#Habil_Mov OR #Mar_Aux)) OR (NOT #iOrdMar AND #iConfMar),
                           PT := #iTConf_Fall);
   #oFall_CTC := #IEC_Timer_0_Instance_1.Q;
   #Fall_CTC_Aux := #IEC_Timer_0_Instance_1.Q;
END_REGION

REGION Network 4: Warning Contactor
   #IEC_Timer_0_Instance.TON(IN := ((#iOrdMar AND NOT #iConfMar AND NOT #Fall_GMT_Aux AND (#Habil_Mov OR #Mar_Aux)) OR (NOT #iOrdMar AND #iConfMar)) AND NOT #Fall_CTC_Aux,
                           PT := #iTConf_Warn);
   #oWarning_CTC := #IEC_Timer_0_Instance.Q;
END_REGION

REGION Network 5: Marcha
   RUNG wire#powerrail
      Contact( #iOrdMar )
      I_Contact( #Fall_GMT_Aux )
      I_Contact( #Fall_CTC_Aux )
      wire#w1
      Contact( #Habil_Mov )
      wire#w2
      Coil( #oMarcha )
   END_RUNG
   RUNG wire#w1
      Contact( #Mar_Aux )
   END_RUNG wire#w2
   RUNG wire#w2
      Coil( #Mar_Aux )
   END_RUNG
   // the same network as SCL:
   #oMarcha := #iOrdMar AND NOT #Fall_GMT_Aux AND NOT #Fall_CTC_Aux AND (#Habil_Mov OR #Mar_Aux);
   #Mar_Aux := #oMarcha;
END_REGION
END_FUNCTION_BLOCK

FUNCTION_BLOCK "FB_VLV_2_POS"   // FB6, LAD
{ S7_Optimized_Access := 'FALSE' }
VERSION : 0.1
   VAR_INPUT
      Ir_Pos_1 : Bool;   // Comando Mover Cilindro a Posición 1, activar constantemente
      Ir_Pos_2 : Bool;   // Comando Mover Cilindro a Posición 2, activar constantemente
      Conf_Pos_1 : Bool;   // Confirmación Cilindro en Posición 1
      Conf_Pos_2 : Bool;   // Confirmación Cilindro en Posición 2
      T_Conf : Time := T#10s;   // Tiempo admisible para confirmación de posición
      T_ON : Time;   // Duración accionamiento salida [0 = constantemente]
   END_VAR
   VAR_OUTPUT
      Pos_1 : Bool;   // Orden Mover Cilindro a Posición 1
      Pos_2 : Bool;   // Orden Mover Cilindro a Posición 2
      ERROR : Int;   // 0 = Sin Error, 1 = Error Programación, 2 = Error Doble Confirmación, 3 = Error Confirmación Pos_1, 4 = Error Confirmación Pos_2, 5 = Sin Confirmaciones
   END_VAR
   VAR
      IEC_Timer_0_Instance : IEC_TIMER;
      IEC_Timer_0_Instance_1 : IEC_TIMER;
      IEC_Timer_0_Instance_2 : IEC_TIMER;
      IEC_Timer_0_Instance_3 : IEC_TIMER;
      IEC_Timer_0_Instance_4 : IEC_TIMER;
   END_VAR
   VAR_TEMP
      Aux_1 : Bool;   // Auxiliar 1
      Aux_2 : Bool;   // Auxiliar 2
      Aux_ERROR : Int;   // Auxiliar ERROR
   END_VAR
BEGIN

REGION Network 1: Auxiliar 1
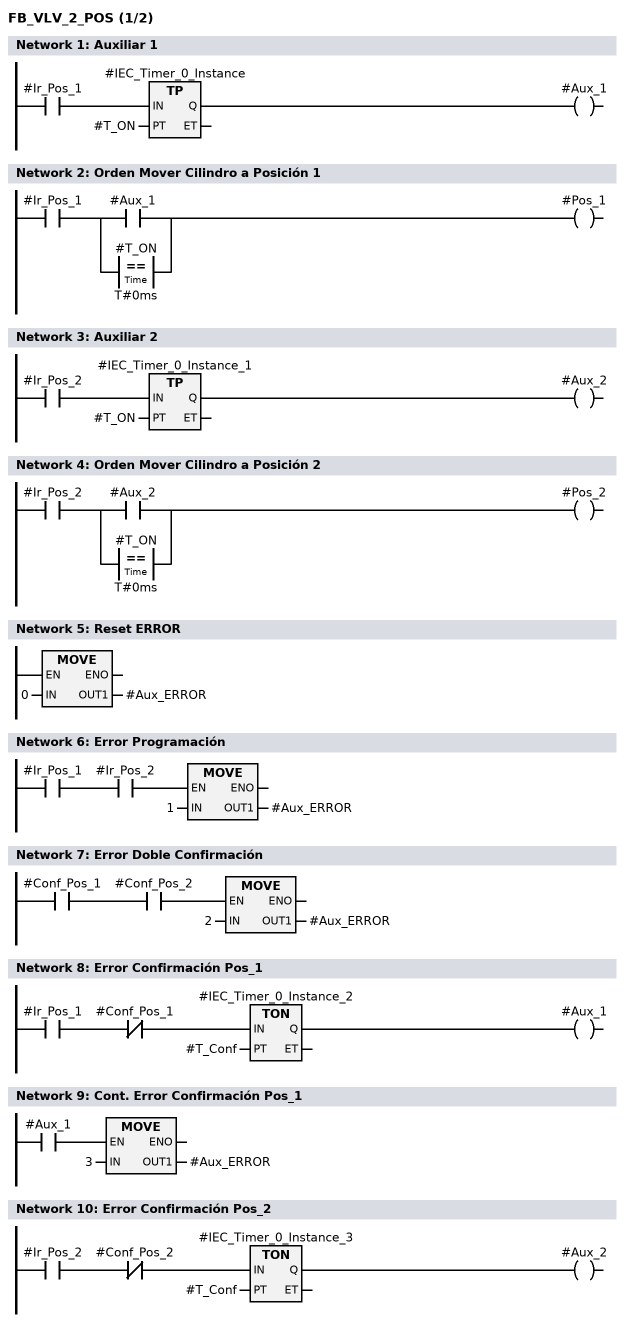
   #IEC_Timer_0_Instance.TP(IN := #Ir_Pos_1, PT := #T_ON);
   #Aux_1 := #IEC_Timer_0_Instance.Q;
END_REGION

REGION Network 2: Orden Mover Cilindro a Posición 1
   RUNG wire#powerrail
      Contact( #Ir_Pos_1 )
      wire#w1
      Contact( #Aux_1 )
      wire#w2
      Coil( #Pos_1 )
   END_RUNG
   RUNG wire#w1
      { S7_Templates := "SrcType := Time" } EQ_Contact(in1 := #T_ON, in2 := T#0ms)
   END_RUNG wire#w2
   // the same network as SCL:
   #Pos_1 := #Ir_Pos_1 AND (#Aux_1 OR (#T_ON = T#0ms));
END_REGION

REGION Network 3: Auxiliar 2
   #IEC_Timer_0_Instance_1.TP(IN := #Ir_Pos_2, PT := #T_ON);
   #Aux_2 := #IEC_Timer_0_Instance_1.Q;
END_REGION

REGION Network 4: Orden Mover Cilindro a Posición 2
   RUNG wire#powerrail
      Contact( #Ir_Pos_2 )
      wire#w1
      Contact( #Aux_2 )
      wire#w2
      Coil( #Pos_2 )
   END_RUNG
   RUNG wire#w1
      { S7_Templates := "SrcType := Time" } EQ_Contact(in1 := #T_ON, in2 := T#0ms)
   END_RUNG wire#w2
   // the same network as SCL:
   #Pos_2 := #Ir_Pos_2 AND (#Aux_2 OR (#T_ON = T#0ms));
END_REGION

REGION Network 5: Reset ERROR
   RUNG wire#powerrail
      { S7_GenerateENO := "TRUE" } Move(in := 0, out1 => #Aux_ERROR)
   END_RUNG
   // the same network as SCL:
   #Aux_ERROR := 0;
END_REGION

REGION Network 6: Error Programación
   RUNG wire#powerrail
      Contact( #Ir_Pos_1 )
      Contact( #Ir_Pos_2 )
      { S7_GenerateENO := "TRUE" } Move(in := 1, out1 => #Aux_ERROR)
   END_RUNG
   // the same network as SCL:
   IF #Ir_Pos_1 AND #Ir_Pos_2 THEN #Aux_ERROR := 1; END_IF;
END_REGION

REGION Network 7: Error Doble Confirmación
   RUNG wire#powerrail
      Contact( #Conf_Pos_1 )
      Contact( #Conf_Pos_2 )
      { S7_GenerateENO := "TRUE" } Move(in := 2, out1 => #Aux_ERROR)
   END_RUNG
   // the same network as SCL:
   IF #Conf_Pos_1 AND #Conf_Pos_2 THEN #Aux_ERROR := 2; END_IF;
END_REGION

REGION Network 8: Error Confirmación Pos_1
   #IEC_Timer_0_Instance_2.TON(IN := #Ir_Pos_1 AND NOT #Conf_Pos_1, PT := #T_Conf);
   #Aux_1 := #IEC_Timer_0_Instance_2.Q;
END_REGION

REGION Network 9: Cont. Error Confirmación Pos_1
   RUNG wire#powerrail
      Contact( #Aux_1 )
      { S7_GenerateENO := "TRUE" } Move(in := 3, out1 => #Aux_ERROR)
   END_RUNG
   // the same network as SCL:
   IF #Aux_1 THEN #Aux_ERROR := 3; END_IF;
END_REGION

REGION Network 10: Error Confirmación Pos_2
   #IEC_Timer_0_Instance_3.TON(IN := #Ir_Pos_2 AND NOT #Conf_Pos_2, PT := #T_Conf);
   #Aux_2 := #IEC_Timer_0_Instance_3.Q;
END_REGION

REGION Network 11: Cont. Error Confirmación Pos_2
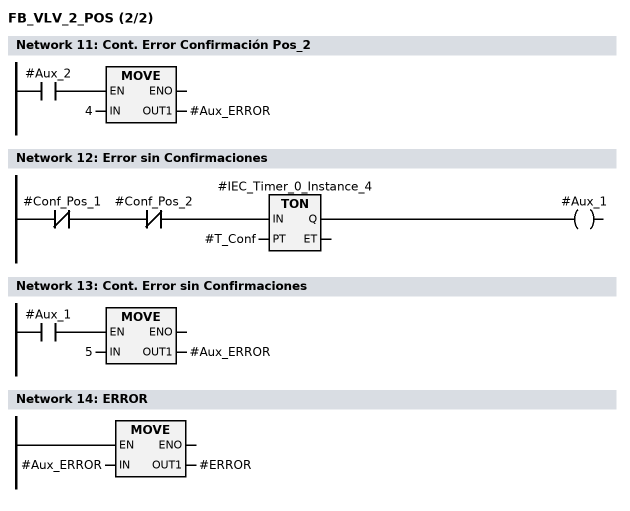
   RUNG wire#powerrail
      Contact( #Aux_2 )
      { S7_GenerateENO := "TRUE" } Move(in := 4, out1 => #Aux_ERROR)
   END_RUNG
   // the same network as SCL:
   IF #Aux_2 THEN #Aux_ERROR := 4; END_IF;
END_REGION

REGION Network 12: Error sin Confirmaciones
   #IEC_Timer_0_Instance_4.TON(IN := NOT #Conf_Pos_1 AND NOT #Conf_Pos_2, PT := #T_Conf);
   #Aux_1 := #IEC_Timer_0_Instance_4.Q;
END_REGION

REGION Network 13: Cont. Error sin Confirmaciones
   RUNG wire#powerrail
      Contact( #Aux_1 )
      { S7_GenerateENO := "TRUE" } Move(in := 5, out1 => #Aux_ERROR)
   END_RUNG
   // the same network as SCL:
   IF #Aux_1 THEN #Aux_ERROR := 5; END_IF;
END_REGION

REGION Network 14: ERROR
   RUNG wire#powerrail
      { S7_GenerateENO := "TRUE" } Move(in := #Aux_ERROR, out1 => #ERROR)
   END_RUNG
   // the same network as SCL:
   #ERROR := #Aux_ERROR;
END_REGION
END_FUNCTION_BLOCK

FUNCTION "MAQ_EST_32" : Void   // FC7, SCL
TITLE = Máquina de Estados 32
{ S7_Optimized_Access := 'TRUE' }
AUTHOR : FRD
FAMILY : MTA
NAME : MaqEst32
VERSION : 1.0
// KNOW_HOW_PROTECT  Máquina de estados de hasta 32 estados.
   VAR_INPUT
      Concatenadoras : DWord;   // Próximo estado de transición normal
      Prioritarias : DWord;   // Próximo estado de transición forzada
   END_VAR
   VAR_OUTPUT
      Error_Concatenadoras : Bool;   // Error en la programación de las Concatenadoras
      Error_Prioritarias : Bool;   // Error en la programación de las Prioritarias
   END_VAR
   VAR_IN_OUT
      Estado : DWord;   // Estado actual
   END_VAR
   VAR_TEMP
      Concat_Int : Int;   // Auxiliar INT para verificar las Concatenadoras
      Priorit_Int : Int;   // Auxiliar INT para verificar las Prioritarias
      Concat_Dword : DWord;   // Auxiliar DWORD para verificar las Concatenadoras
      Priorit_Dword : DWord;   // Auxiliar DWORD para verificar las Prioritarias
      Activar_Concat : Bool;   // Bit que indica Concatenadoras correctas
      Activar_Priorit : Bool;   // Bit que indica Prioritarias correctas
      Falla_Concat : Bool;   // Bit que indica falla en Concatenadoras
      Falla_Priorit : Bool;   // Bit que indica falla en Prioritarias
   END_VAR
BEGIN
   #Falla_Concat := 0;
   #Activar_Concat := 0;
   #Falla_Priorit := 0;
   #Activar_Priorit := 0; 
   #Error_Concatenadoras := 0;
   #Error_Prioritarias := 0;

   IF #Concatenadoras <> 0 THEN     //Evaluar Concatenadoras si son distintas de "0"

    #Concat_Int := ENCO(IN := #Concatenadoras );  //Convierte posición_DWORD en INT (0 a 31), lee el LSb

    #Concat_Dword := DECO(IN := INT_TO_UINT(#Concat_Int));//Convierte INT en posición_DWORD (1 a 32)

    IF #Concatenadoras = #Concat_Dword THEN  //Si son iguales, había sólo un bit en "1"

     #Activar_Concat := 1;    //Concatenadora correcta

    ELSE

     #Falla_Concat := 1;    //Falla en Concatenadora

    END_IF;

   END_IF;

   IF #Prioritarias <> 0 THEN     //Evaluar Prioritarias si son distintas de "0"

    #Priorit_Int := ENCO(IN := #Prioritarias);  //Convierte posición_DWORD en INT (0 a 31), lee el LSb

    #Priorit_Dword := DECO(IN := INT_TO_UINT(#Priorit_Int));//Convierte INT en posición_DWORD (1 a 32)

    IF #Prioritarias = #Priorit_Dword THEN  //Si son iguales, había sólo un bit en "1"

     #Activar_Priorit := 1;   //Prioritaria correcta

    ELSE

     #Falla_Priorit := 1;    //Falla en Prioritaria

    END_IF;

   END_IF;

   IF NOT(#Falla_Priorit OR #Falla_Concat) THEN  //Si no hay falla de Prioritaria ni de Concatenadora

    IF #Activar_Priorit THEN    //Si hay que asignar Prioritarias

     #Estado := #Prioritarias;

    ELSE

     IF #Activar_Concat THEN   //Si hay que asignar Concatenadoras

      #Estado := #Concatenadoras;

     END_IF;

    END_IF;

   ELSE

    IF #Falla_Concat THEN     //Si hay falla de Concatenadoras

     #Error_Concatenadoras := 1;    //Activar Error_Concatenadoras

    END_IF;

    IF #Falla_Priorit THEN    //Si hay falla de Prioritarias

     #Error_Prioritarias := 1;    //Activar Error_Prioritarias

    END_IF;

   END_IF;
END_FUNCTION

// folder: INCIDENTES

FUNCTION_BLOCK "FB_INC_GENERAL"   // FB500, LAD
TITLE = ALARMAS GENERAL
{ S7_Optimized_Access := 'FALSE' }
VERSION : 0.1
   VAR
      Alarma_On : Bool;
   END_VAR
BEGIN

REGION Network 1: Marca 1 - Protecciones abiertas
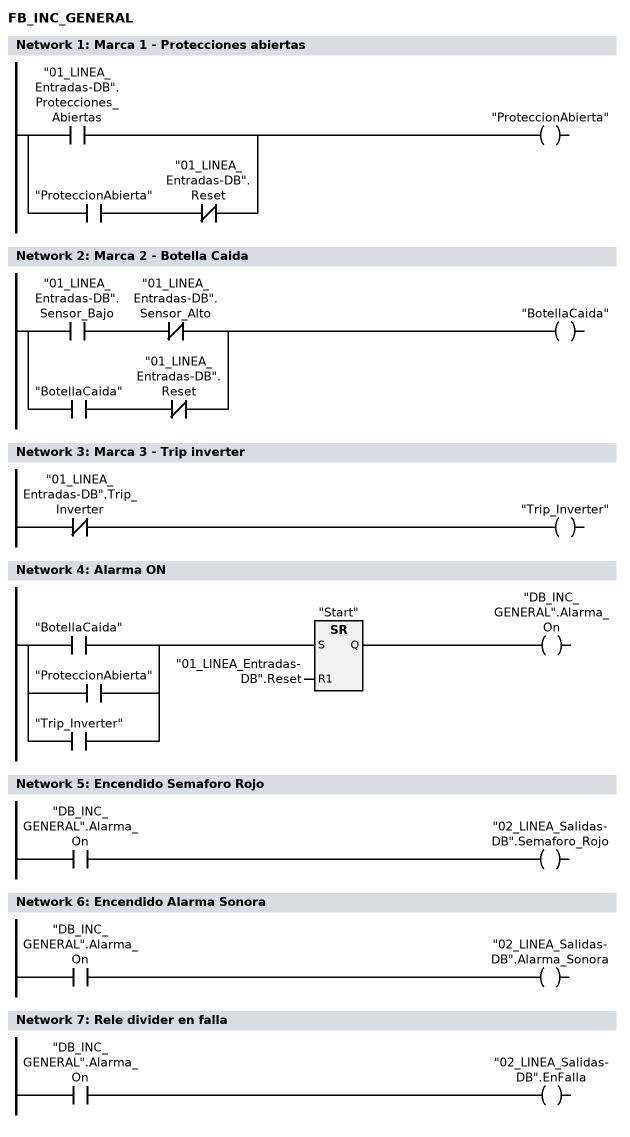
   RUNG wire#powerrail
      Contact( "01_LINEA_Entradas-DB".Protecciones_Abiertas )
      wire#w1
      Coil( "ProteccionAbierta" )
   END_RUNG
   RUNG wire#powerrail
      Contact( "ProteccionAbierta" )
      I_Contact( "01_LINEA_Entradas-DB".Reset )
   END_RUNG wire#w1
   // the same network as SCL:
   "ProteccionAbierta" := "01_LINEA_Entradas-DB".Protecciones_Abiertas OR ("ProteccionAbierta" AND NOT "01_LINEA_Entradas-DB".Reset);
END_REGION

REGION Network 2: Marca 2 - Botella Caida
   RUNG wire#powerrail
      Contact( "01_LINEA_Entradas-DB".Sensor_Bajo )
      I_Contact( "01_LINEA_Entradas-DB".Sensor_Alto )
      wire#w1
      Coil( "BotellaCaida" )
   END_RUNG
   RUNG wire#powerrail
      Contact( "BotellaCaida" )
      I_Contact( "01_LINEA_Entradas-DB".Reset )
   END_RUNG wire#w1
   // the same network as SCL:
   "BotellaCaida" := ("01_LINEA_Entradas-DB".Sensor_Bajo AND NOT "01_LINEA_Entradas-DB".Sensor_Alto) OR ("BotellaCaida" AND NOT "01_LINEA_Entradas-DB".Reset);
END_REGION

REGION Network 3: Marca 3 - Trip inverter
   RUNG wire#powerrail
      I_Contact( "01_LINEA_Entradas-DB".Trip_Inverter )
      Coil( "Trip_Inverter" )
   END_RUNG
   // the same network as SCL:
   "Trip_Inverter" := NOT "01_LINEA_Entradas-DB".Trip_Inverter;
END_REGION

REGION Network 4: Alarma ON
   RUNG wire#powerrail
      Contact( "BotellaCaida" )
      wire#w1
      S_SR(operand := "Start", r1 := "01_LINEA_Entradas-DB".Reset)
      Coil( "DB_INC_GENERAL".Alarma_On )
   END_RUNG
   RUNG wire#powerrail
      Contact( "ProteccionAbierta" )
   END_RUNG wire#w1
   RUNG wire#powerrail
      Contact( "Trip_Inverter" )
   END_RUNG wire#w1
   // the same network as SCL:
   IF "BotellaCaida" OR "ProteccionAbierta" OR "Trip_Inverter" THEN
       "Start" := TRUE;   // SR flip-flop
   END_IF;
   IF "01_LINEA_Entradas-DB".Reset THEN "Start" := FALSE; END_IF;
   "DB_INC_GENERAL".Alarma_On := "Start";
END_REGION

REGION Network 5: Encendido Semaforo Rojo
   RUNG wire#powerrail
      Contact( "DB_INC_GENERAL".Alarma_On )
      Coil( "02_LINEA_Salidas-DB".Semaforo_Rojo )
   END_RUNG
   // the same network as SCL:
   "02_LINEA_Salidas-DB".Semaforo_Rojo := "DB_INC_GENERAL".Alarma_On;
END_REGION

REGION Network 6: Encendido Alarma Sonora
   RUNG wire#powerrail
      Contact( "DB_INC_GENERAL".Alarma_On )
      Coil( "02_LINEA_Salidas-DB".Alarma_Sonora )
   END_RUNG
   // the same network as SCL:
   "02_LINEA_Salidas-DB".Alarma_Sonora := "DB_INC_GENERAL".Alarma_On;
END_REGION

REGION Network 7: Rele divider en falla
   RUNG wire#powerrail
      Contact( "DB_INC_GENERAL".Alarma_On )
      Coil( "02_LINEA_Salidas-DB".EnFalla )
   END_RUNG
   // the same network as SCL:
   "02_LINEA_Salidas-DB".EnFalla := "DB_INC_GENERAL".Alarma_On;
END_REGION
END_FUNCTION_BLOCK